SPLINE
SPL {X  -158.454, Y  +360.384, Z    +0.000, E1  +340.634, E3 -463508.318}
SPL {X  -159.737, Y  +373.507, Z    +0.000, E1  +349.689, E3 -463530.353}
SPL {X  -159.990, Y  +382.574, Z    +0.000, E1  +355.537, E3 -463537.041}
SPL {X  -159.990, Y  +389.909, Z    +0.000, E1  +360.662, E3 -463541.055}
SPL {X  -159.990, Y  +396.289, Z    +0.000, E1  +365.500, E3 -463544.835}
SPL {X  -159.990, Y  +407.941, Z    +0.000, E1  +374.126, E3 -463556.172}
SPL {X  -159.990, Y  +418.671, Z    +0.000, E1  +379.855, E3 -463575.589}
SPL {X  -159.990, Y  +429.878, Z    +0.000, E1  +383.330, E3 -463605.644}
SPL {X  -159.990, Y  +432.103, Z    +0.000, E1  +383.301, E3 -463616.662}
SPL {X  -159.990, Y  +434.188, Z    +0.000, E1  +383.325, E3 -463626.859}
SPL {X  -159.990, Y  +436.320, Z    +0.000, E1  +383.304, E3 -463637.411}
SPL {X  -159.990, Y  +439.169, Z    +0.000, E1  +383.353, E3 -463651.329}
SPL {X  -159.990, Y  +442.945, Z    +0.000, E1  +383.339, E3 -463669.946}
SPL {X  -159.990, Y  +446.037, Z    +0.000, E1  +383.324, E3 -463685.196}
SPL {X  -159.990, Y  +448.341, Z    +0.000, E1  +383.317, E3 -463696.514}
SPL {X  -159.990, Y  +450.345, Z    +0.000, E1  +383.316, E3 -463706.392}
SPL {X  -159.990, Y  +452.828, Z    +0.000, E1  +383.330, E3 -463718.591}
SPL {X  -159.990, Y  +456.338, Z    +0.000, E1  +383.359, E3 -463735.784}
SPL {X  -159.990, Y  +459.480, Z    +0.000, E1  +383.323, E3 -463751.325}
SPL {X  -159.990, Y  +461.803, Z    +0.000, E1  +383.322, E3 -463762.760}
SPL {X  -159.990, Y  +464.971, Z    +0.000, E1  +383.357, E3 -463778.266}
SPL {X  -159.990, Y  +467.934, Z    +0.000, E1  +383.321, E3 -463792.923}
SPL {X  -159.990, Y  +469.939, Z    +0.000, E1  +383.319, E3 -463802.785}
SPL {X  -159.990, Y  +472.144, Z    +0.000, E1  +383.327, E3 -463813.636}
SPL {X  -159.990, Y  +474.994, Z    +0.000, E1  +383.334, E3 -463827.684}
SPL {X  -159.990, Y  +477.323, Z    +0.000, E1  +383.307, E3 -463839.199}
SPL {X  -159.990, Y  +479.553, Z    +0.000, E1  +383.328, E3 -463850.134}
SPL {X  -159.990, Y  +482.799, Z    +0.000, E1  +383.343, E3 -463866.074}
SPL {X  -159.990, Y  +485.299, Z    +0.000, E1  +383.310, E3 -463878.459}
SPL {X  -159.990, Y  +488.031, Z    +0.000, E1  +383.345, E3 -463891.838}
SPL {X  -159.990, Y  +491.121, Z    +0.000, E1  +383.323, E3 -463907.083}
SPL {X  -159.990, Y  +493.610, Z    +0.000, E1  +383.323, E3 -463919.336}
SPL {X  -159.990, Y  +495.794, Z    +0.000, E1  +383.312, E3 -463930.110}
SPL {X  -159.990, Y  +497.668, Z    +0.000, E1  +383.317, E3 -463939.319}
SPL {X  -159.990, Y  +499.995, Z    +0.000, E1  +383.324, E3 -463950.757}
SPL {X  -159.990, Y  +502.341, Z    +0.000, E1  +383.320, E3 -463962.316}
SPL {X  -159.990, Y  +504.419, Z    +0.000, E1  +383.313, E3 -463972.558}
SPL {X  -159.990, Y  +507.187, Z    +0.000, E1  +383.346, E3 -463986.111}
SPL {X  -159.990, Y  +510.344, Z    +0.000, E1  +383.327, E3 -464001.696}
SPL {X  -159.990, Y  +512.484, Z    +0.000, E1  +383.309, E3 -464012.269}
SPL {X  -159.990, Y  +514.016, Z    +0.000, E1  +383.308, E3 -464019.817}
SPL {X  -159.990, Y  +516.195, Z    +0.000, E1  +383.325, E3 -464030.505}
SPL {X  -159.990, Y  +518.925, Z    +0.000, E1  +383.333, E3 -464043.868}
SPL {X  -159.990, Y  +521.408, Z    +0.000, E1  +383.329, E3 -464056.077}
SPL {X  -159.990, Y  +523.942, Z    +0.000, E1  +383.333, E3 -464068.570}
SPL {X  -159.990, Y  +526.221, Z    +0.000, E1  +383.314, E3 -464079.846}
SPL {X  -159.990, Y  +527.834, Z    +0.000, E1  +383.311, E3 -464087.796}
SPL {X  -159.990, Y  +529.993, Z    +0.000, E1  +383.329, E3 -464098.372}
SPL {X  -159.990, Y  +532.441, Z    +0.000, E1  +383.322, E3 -464110.423}
SPL {X  -159.990, Y  +534.618, Z    +0.000, E1  +383.322, E3 -464121.156}
SPL {X  -159.990, Y  +537.024, Z    +0.000, E1  +383.321, E3 -464133.018}
SPL {X  -159.990, Y  +539.129, Z    +0.000, E1  +383.310, E3 -464143.401}
SPL {X  -159.990, Y  +541.183, Z    +0.000, E1  +383.319, E3 -464153.498}
SPL {X  -159.990, Y  +543.647, Z    +0.000, E1  +383.325, E3 -464165.601}
SPL {X  -159.990, Y  +545.957, Z    +0.000, E1  +383.318, E3 -464176.981}
SPL {X  -159.990, Y  +548.912, Z    +0.000, E1  +383.354, E3 -464191.441}
SPL {X  -159.990, Y  +551.655, Z    +0.000, E1  +383.320, E3 -464205.016}
SPL {X  -159.990, Y  +553.711, Z    +0.000, E1  +383.317, E3 -464215.137}
SPL {X  -159.990, Y  +556.481, Z    +0.000, E1  +383.354, E3 -464228.699}
SPL {X  -159.990, Y  +559.475, Z    +0.000, E1  +383.321, E3 -464243.505}
SPL {X  -159.990, Y  +561.830, Z    +0.000, E1  +383.325, E3 -464255.089}
SPL {X  -159.990, Y  +564.273, Z    +0.000, E1  +383.325, E3 -464267.113}
SPL {X  -159.990, Y  +566.342, Z    +0.000, E1  +383.314, E3 -464277.318}
SPL {X  -159.990, Y  +568.184, Z    +0.000, E1  +383.317, E3 -464286.379}
SPL {X  -159.990, Y  +570.314, Z    +0.000, E1  +383.326, E3 -464296.841}
SPL {X  -159.990, Y  +573.444, Z    +0.000, E1  +383.356, E3 -464312.181}
SPL {X  -159.990, Y  +577.161, Z    +0.000, E1  +383.346, E3 -464330.505}
SPL {X  -159.990, Y  +580.840, Z    +0.000, E1  +383.355, E3 -464348.554}
SPL {X  -159.990, Y  +583.973, Z    +0.000, E1  +383.332, E3 -464364.016}
SPL {X  -159.990, Y  +586.020, Z    +0.000, E1  +383.323, E3 -464374.099}
SPL {X  -159.990, Y  +587.711, Z    +0.000, E1  +383.318, E3 -464382.439}
SPL {X  -159.990, Y  +589.763, Z    +0.000, E1  +383.328, E3 -464392.515}
SPL {X  -159.990, Y  +591.698, Z    +0.000, E1  +383.324, E3 -464402.000}
SPL {X  -159.990, Y  +593.847, Z    +0.000, E1  +383.340, E3 -464412.531}
SPL {X  -159.990, Y  +597.018, Z    +0.000, E1  +383.367, E3 -464428.063}
SPL {X  -159.990, Y  +599.887, Z    +0.000, E1  +383.341, E3 -464442.167}
SPL {X  -159.990, Y  +601.949, Z    +0.000, E1  +383.344, E3 -464452.294}
SPL {X  -159.990, Y  +605.106, Z    +0.000, E1  +383.383, E3 -464467.740}
SPL {X  -159.990, Y  +608.111, Z    +0.000, E1  +383.342, E3 -464482.591}
SPL {X  -159.990, Y  +610.073, Z    +0.000, E1  +383.343, E3 -464492.249}
SPL {X  -159.990, Y  +612.330, Z    +0.000, E1  +383.340, E3 -464503.376}
SPL {X  -159.990, Y  +615.036, Z    +0.000, E1  +383.353, E3 -464516.663}
SPL {X  -159.990, Y  +618.481, Z    +0.000, E1  +383.366, E3 -464533.601}
SPL {X  -159.990, Y  +621.517, Z    +0.000, E1  +383.337, E3 -464548.584}
SPL {X  -159.990, Y  +623.764, Z    +0.000, E1  +383.335, E3 -464559.635}
SPL {X  -159.990, Y  +626.608, Z    +0.000, E1  +383.361, E3 -464573.560}
SPL {X  -159.990, Y  +630.271, Z    +0.000, E1  +383.375, E3 -464591.521}
SPL {X  -159.990, Y  +633.318, Z    +0.000, E1  +383.339, E3 -464606.598}
SPL {X  -159.990, Y  +635.650, Z    +0.000, E1  +383.339, E3 -464618.069}
SPL {X  -159.990, Y  +638.406, Z    +0.000, E1  +383.354, E3 -464631.636}
SPL {X  -159.990, Y  +641.831, Z    +0.000, E1  +383.342, E3 -464648.583}
SPL {X  -159.990, Y  +644.884, Z    +0.000, E1  +383.324, E3 -464663.670}
SPL {X  -159.990, Y  +647.550, Z    +0.000, E1  +383.318, E3 -464676.837}
SPL {X  -159.990, Y  +650.790, Z    +0.000, E1  +383.346, E3 -464692.704}
SPL {X  -159.990, Y  +654.543, Z    +0.000, E1  +383.348, E3 -464711.157}
SPL {X  -159.990, Y  +658.319, Z    +0.000, E1  +383.349, E3 -464729.746}
SPL {X  -159.990, Y  +661.392, Z    +0.000, E1  +383.318, E3 -464744.949}
SPL {X  -159.990, Y  +663.662, Z    +0.000, E1  +383.322, E3 -464756.073}
SPL {X  -159.990, Y  +665.964, Z    +0.000, E1  +383.328, E3 -464767.364}
SPL {X  -159.990, Y  +667.870, Z    +0.000, E1  +383.320, E3 -464776.771}
SPL {X  -159.990, Y  +669.861, Z    +0.000, E1  +383.321, E3 -464786.572}
SPL {X  -159.983, Y  +672.946, Z    +0.000, E1  +383.359, E3 -464801.681}
SPL {X  -159.924, Y  +676.110, Z    +0.000, E1  +383.320, E3 -464817.380}
SPL {X  -159.801, Y  +679.265, Z    +0.000, E1  +383.327, E3 -464832.999}
SPL {X  -159.626, Y  +682.287, Z    +0.000, E1  +383.280, E3 -464848.097}
SPL {X  -159.462, Y  +684.486, Z    +0.000, E1  +383.258, E3 -464859.097}
SPL {X  -159.289, Y  +686.457, Z    +0.000, E1  +383.223, E3 -464869.007}
SPL {X  -159.052, Y  +688.801, Z    +0.000, E1  +383.217, E3 -464880.742}
SPL {X  -158.770, Y  +691.222, Z    +0.000, E1  +383.158, E3 -464893.000}
SPL {X  -158.553, Y  +692.896, Z    +0.000, E1  +383.130, E3 -464901.465}
ENDSPLINE

SPLINE
SPL {X  -159.063, Y  +688.696, Z    +0.000, E1  +377.094, E3 -464939.586}
SPL {X  -159.987, Y  +672.488, Z    +0.000, E1  +365.638, E3 -464963.651}
SPL {X  -159.990, Y  +663.928, Z    +0.000, E1  +359.662, E3 -464969.445}
SPL {X  -159.990, Y  +658.009, Z    +0.000, E1  +355.226, E3 -464973.145}
SPL {X  -159.990, Y  +651.879, Z    +0.000, E1  +350.548, E3 -464978.208}
SPL {X  -159.990, Y  +637.832, Z    +0.000, E1  +341.694, E3 -464995.799}
SPL {X  -159.990, Y  +626.634, Z    +0.000, E1  +337.968, E3 -465026.652}
SPL {X  -159.990, Y  +624.622, Z    +0.000, E1  +337.980, E3 -465037.235}
SPL {X  -159.990, Y  +622.489, Z    +0.000, E1  +337.969, E3 -465048.402}
SPL {X  -159.990, Y  +619.955, Z    +0.000, E1  +337.968, E3 -465061.692}
SPL {X  -159.990, Y  +617.386, Z    +0.000, E1  +337.968, E3 -465075.167}
SPL {X  -159.990, Y  +614.863, Z    +0.000, E1  +337.969, E3 -465088.399}
SPL {X  -159.990, Y  +612.600, Z    +0.000, E1  +337.975, E3 -465100.283}
SPL {X  -159.990, Y  +610.646, Z    +0.000, E1  +337.979, E3 -465110.540}
SPL {X  -159.990, Y  +608.810, Z    +0.000, E1  +337.977, E3 -465120.173}
SPL {X  -159.990, Y  +606.481, Z    +0.000, E1  +337.967, E3 -465132.349}
SPL {X  -159.990, Y  +603.419, Z    +0.000, E1  +337.936, E3 -465148.288}
SPL {X  -159.990, Y  +600.642, Z    +0.000, E1  +337.968, E3 -465162.918}
SPL {X  -159.990, Y  +598.568, Z    +0.000, E1  +337.954, E3 -465173.710}
SPL {X  -159.990, Y  +595.493, Z    +0.000, E1  +337.930, E3 -465189.794}
SPL {X  -159.990, Y  +592.865, Z    +0.000, E1  +337.964, E3 -465203.622}
SPL {X  -159.990, Y  +590.803, Z    +0.000, E1  +337.954, E3 -465214.413}
SPL {X  -159.990, Y  +588.288, Z    +0.000, E1  +337.950, E3 -465227.577}
SPL {X  -159.990, Y  +586.040, Z    +0.000, E1  +337.954, E3 -465239.322}
SPL {X  -159.990, Y  +584.080, Z    +0.000, E1  +337.953, E3 -465249.582}
SPL {X  -159.990, Y  +581.924, Z    +0.000, E1  +337.949, E3 -465260.883}
SPL {X  -159.990, Y  +579.673, Z    +0.000, E1  +337.950, E3 -465272.681}
SPL {X  -159.990, Y  +576.961, Z    +0.000, E1  +337.936, E3 -465286.860}
SPL {X  -159.990, Y  +574.188, Z    +0.000, E1  +337.947, E3 -465301.407}
SPL {X  -159.990, Y  +571.954, Z    +0.000, E1  +337.959, E3 -465313.165}
SPL {X  -159.990, Y  +570.110, Z    +0.000, E1  +337.958, E3 -465322.815}
SPL {X  -159.990, Y  +568.165, Z    +0.000, E1  +337.957, E3 -465332.995}
SPL {X  -159.990, Y  +565.292, Z    +0.000, E1  +337.922, E3 -465347.973}
SPL {X  -159.990, Y  +562.598, Z    +0.000, E1  +337.958, E3 -465362.184}
SPL {X  -159.990, Y  +560.652, Z    +0.000, E1  +337.962, E3 -465372.396}
SPL {X  -159.990, Y  +558.143, Z    +0.000, E1  +337.928, E3 -465385.428}
SPL {X  -159.990, Y  +555.329, Z    +0.000, E1  +337.943, E3 -465400.172}
SPL {X  -159.990, Y  +553.115, Z    +0.000, E1  +337.946, E3 -465411.778}
SPL {X  -159.990, Y  +550.886, Z    +0.000, E1  +337.944, E3 -465423.459}
SPL {X  -159.990, Y  +548.568, Z    +0.000, E1  +337.944, E3 -465435.580}
SPL {X  -159.990, Y  +545.859, Z    +0.000, E1  +337.926, E3 -465449.730}
SPL {X  -159.990, Y  +542.390, Z    +0.000, E1  +337.914, E3 -465467.900}
SPL {X  -159.990, Y  +539.341, Z    +0.000, E1  +337.944, E3 -465483.922}
SPL {X  -159.990, Y  +536.935, Z    +0.000, E1  +337.942, E3 -465496.511}
SPL {X  -159.990, Y  +534.656, Z    +0.000, E1  +337.946, E3 -465508.455}
SPL {X  -159.990, Y  +532.453, Z    +0.000, E1  +337.944, E3 -465519.982}
SPL {X  -159.990, Y  +530.660, Z    +0.000, E1  +337.952, E3 -465529.385}
SPL {X  -159.990, Y  +528.702, Z    +0.000, E1  +337.939, E3 -465539.598}
SPL {X  -159.990, Y  +525.760, Z    +0.000, E1  +337.914, E3 -465554.939}
SPL {X  -159.990, Y  +522.838, Z    +0.000, E1  +337.933, E3 -465570.306}
SPL {X  -159.990, Y  +519.698, Z    +0.000, E1  +337.916, E3 -465586.689}
SPL {X  -159.990, Y  +517.251, Z    +0.000, E1  +337.946, E3 -465599.549}
SPL {X  -159.990, Y  +515.568, Z    +0.000, E1  +338.084, E3 -465609.646}
ENDSPLINE

SPLINE
SPL {X  -159.990, Y  +517.293, Z    +0.000, E1  +340.923, E3 -465625.944}
ENDSPLINE

SPLINE
SPL {X  -159.990, Y  +512.548, Z    +0.000, E1  +339.587, E3 -465641.519}
SPL {X  -159.990, Y  +508.660, Z    +0.000, E1  +338.515, E3 -465653.573}
SPL {X  -159.990, Y  +503.499, Z    +0.000, E1  +337.116, E3 -465668.653}
SPL {X  -159.990, Y  +498.406, Z    +0.000, E1  +335.789, E3 -465682.685}
SPL {X  -159.990, Y  +494.693, Z    +0.000, E1  +334.929, E3 -465693.153}
SPL {X  -159.990, Y  +491.649, Z    +0.000, E1  +334.596, E3 -465704.355}
SPL {X  -159.990, Y  +488.807, Z    +0.000, E1  +334.603, E3 -465717.080}
SPL {X  -159.990, Y  +486.070, Z    +0.000, E1  +334.601, E3 -465729.311}
SPL {X  -159.990, Y  +483.747, Z    +0.000, E1  +334.616, E3 -465739.724}
SPL {X  -159.990, Y  +481.038, Z    +0.000, E1  +334.588, E3 -465751.779}
SPL {X  -159.990, Y  +478.407, Z    +0.000, E1  +334.616, E3 -465763.593}
SPL {X  -159.990, Y  +475.940, Z    +0.000, E1  +334.597, E3 -465774.583}
SPL {X  -159.990, Y  +473.026, Z    +0.000, E1  +334.601, E3 -465787.613}
SPL {X  -159.990, Y  +470.047, Z    +0.000, E1  +334.598, E3 -465800.931}
SPL {X  -159.990, Y  +467.082, Z    +0.000, E1  +334.601, E3 -465814.178}
SPL {X  -159.990, Y  +464.919, Z    +0.000, E1  +334.619, E3 -465823.905}
SPL {X  -159.990, Y  +462.520, Z    +0.000, E1  +334.600, E3 -465834.580}
SPL {X  -159.990, Y  +460.081, Z    +0.000, E1  +334.610, E3 -465845.481}
SPL {X  -159.990, Y  +457.497, Z    +0.000, E1  +334.597, E3 -465857.005}
SPL {X  -159.990, Y  +454.323, Z    +0.000, E1  +334.588, E3 -465871.165}
SPL {X  -159.990, Y  +450.823, Z    +0.000, E1  +334.583, E3 -465886.793}
SPL {X  -159.990, Y  +446.894, Z    +0.000, E1  +334.572, E3 -465904.350}
SPL {X  -159.990, Y  +443.345, Z    +0.000, E1  +334.610, E3 -465920.358}
SPL {X  -159.990, Y  +441.077, Z    +0.000, E1  +334.631, E3 -465930.556}
SPL {X  -159.990, Y  +438.608, Z    +0.000, E1  +334.608, E3 -465941.553}
SPL {X  -159.990, Y  +435.579, Z    +0.000, E1  +334.614, E3 -465955.107}
SPL {X  -159.990, Y  +432.613, Z    +0.000, E1  +334.610, E3 -465968.374}
SPL {X  -159.990, Y  +429.079, Z    +0.000, E1  +334.593, E3 -465984.145}
SPL {X  -159.990, Y  +426.149, Z    +0.000, E1  +334.626, E3 -465997.307}
SPL {X  -159.990, Y  +423.417, Z    +0.000, E1  +334.600, E3 -466009.472}
SPL {X  -159.990, Y  +419.467, Z    +0.000, E1  +334.583, E3 -466027.107}
SPL {X  -159.990, Y  +415.368, Z    +0.000, E1  +334.593, E3 -466045.462}
SPL {X  -159.990, Y  +411.297, Z    +0.000, E1  +334.587, E3 -466063.657}
SPL {X  -159.990, Y  +407.450, Z    +0.000, E1  +334.599, E3 -466080.871}
SPL {X  -159.990, Y  +403.513, Z    +0.000, E1  +334.580, E3 -466098.425}
SPL {X  -159.990, Y  +399.294, Z    +0.000, E1  +334.582, E3 -466117.305}
SPL {X  -159.990, Y  +395.411, Z    +0.000, E1  +334.600, E3 -466134.719}
SPL {X  -159.990, Y  +392.473, Z    +0.000, E1  +334.623, E3 -466147.904}
SPL {X  -159.990, Y  +390.187, Z    +0.000, E1  +334.622, E3 -466158.163}
SPL {X  -159.990, Y  +387.503, Z    +0.000, E1  +334.622, E3 -466170.157}
SPL {X  -159.990, Y  +384.711, Z    +0.000, E1  +334.612, E3 -466182.601}
SPL {X  -159.988, Y  +381.794, Z    +0.000, E1  +334.611, E3 -466195.636}
SPL {X  -159.958, Y  +379.279, Z    +0.000, E1  +334.625, E3 -466206.926}
SPL {X  -159.894, Y  +376.959, Z    +0.000, E1  +334.630, E3 -466217.370}
SPL {X  -159.765, Y  +374.027, Z    +0.000, E1  +334.633, E3 -466230.586}
SPL {X  -159.607, Y  +371.442, Z    +0.000, E1  +334.673, E3 -466242.361}
SPL {X  -159.379, Y  +368.534, Z    +0.000, E1  +334.684, E3 -466255.549}
SPL {X  -159.113, Y  +365.767, Z    +0.000, E1  +334.734, E3 -466268.188}
SPL {X  -158.869, Y  +363.595, Z    +0.000, E1  +334.770, E3 -466278.160}
SPL {X  -158.527, Y  +360.915, Z    +0.000, E1  +334.798, E3 -466290.466}
SPL {X  -158.127, Y  +358.155, Z    +0.000, E1  +334.874, E3 -466303.304}
SPL {X  -158.095, Y  +357.947, Z    +0.000, E1  +338.259, E3 -466334.876}
ENDSPLINE

SPLINE
SPL {X  -158.454, Y  +360.384, Z    +0.000, E1  +340.634, E3 -466347.027}
SPL {X  -159.737, Y  +373.507, Z    +0.000, E1  +349.689, E3 -466369.063}
SPL {X  -159.990, Y  +382.574, Z    +0.000, E1  +355.537, E3 -466375.750}
SPL {X  -159.990, Y  +387.496, Z    +0.000, E1  +358.996, E3 -466378.496}
SPL {X  -159.990, Y  +395.121, Z    +0.000, E1  +364.514, E3 -466382.808}
SPL {X  -159.990, Y  +407.941, Z    +0.000, E1  +374.126, E3 -466394.882}
SPL {X  -159.990, Y  +418.671, Z    +0.000, E1  +379.855, E3 -466414.298}
SPL {X  -159.990, Y  +429.878, Z    +0.000, E1  +383.330, E3 -466444.353}
SPL {X  -159.990, Y  +432.103, Z    +0.000, E1  +383.301, E3 -466455.372}
SPL {X  -159.990, Y  +434.188, Z    +0.000, E1  +383.325, E3 -466465.568}
SPL {X  -159.990, Y  +436.320, Z    +0.000, E1  +383.304, E3 -466476.121}
SPL {X  -159.990, Y  +439.169, Z    +0.000, E1  +383.353, E3 -466490.038}
SPL {X  -159.990, Y  +442.945, Z    +0.000, E1  +383.339, E3 -466508.656}
SPL {X  -159.990, Y  +446.037, Z    +0.000, E1  +383.324, E3 -466523.906}
SPL {X  -159.990, Y  +448.341, Z    +0.000, E1  +383.317, E3 -466535.224}
SPL {X  -159.990, Y  +450.968, Z    +0.000, E1  +383.336, E3 -466548.139}
SPL {X  -159.990, Y  +454.421, Z    +0.000, E1  +383.348, E3 -466565.088}
SPL {X  -159.990, Y  +457.167, Z    +0.000, E1  +383.324, E3 -466578.631}
SPL {X  -159.990, Y  +459.480, Z    +0.000, E1  +383.323, E3 -466590.035}
SPL {X  -159.990, Y  +462.520, Z    +0.000, E1  +383.350, E3 -466604.939}
SPL {X  -159.990, Y  +465.602, Z    +0.000, E1  +383.328, E3 -466620.139}
SPL {X  -159.990, Y  +467.934, Z    +0.000, E1  +383.321, E3 -466631.633}
SPL {X  -159.990, Y  +469.939, Z    +0.000, E1  +383.319, E3 -466641.495}
SPL {X  -159.990, Y  +472.144, Z    +0.000, E1  +383.327, E3 -466652.345}
SPL {X  -159.990, Y  +474.152, Z    +0.000, E1  +383.309, E3 -466662.297}
SPL {X  -159.990, Y  +476.560, Z    +0.000, E1  +383.332, E3 -466674.106}
SPL {X  -159.990, Y  +478.770, Z    +0.000, E1  +383.306, E3 -466685.031}
SPL {X  -159.990, Y  +480.905, Z    +0.000, E1  +383.327, E3 -466695.499}
SPL {X  -159.990, Y  +484.251, Z    +0.000, E1  +383.352, E3 -466711.914}
SPL {X  -159.990, Y  +488.031, Z    +0.000, E1  +383.345, E3 -466730.547}
SPL {X  -159.990, Y  +491.121, Z    +0.000, E1  +383.323, E3 -466745.793}
SPL {X  -159.990, Y  +493.610, Z    +0.000, E1  +383.323, E3 -466758.046}
SPL {X  -159.990, Y  +496.863, Z    +0.000, E1  +383.350, E3 -466774.006}
SPL {X  -159.990, Y  +499.995, Z    +0.000, E1  +383.324, E3 -466789.467}
SPL {X  -159.990, Y  +502.341, Z    +0.000, E1  +383.320, E3 -466801.026}
SPL {X  -159.990, Y  +505.377, Z    +0.000, E1  +383.346, E3 -466815.917}
SPL {X  -159.990, Y  +508.024, Z    +0.000, E1  +383.315, E3 -466828.999}
SPL {X  -159.990, Y  +510.344, Z    +0.000, E1  +383.327, E3 -466840.406}
SPL {X  -159.990, Y  +513.289, Z    +0.000, E1  +383.332, E3 -466854.896}
SPL {X  -159.990, Y  +516.195, Z    +0.000, E1  +383.325, E3 -466869.215}
SPL {X  -159.990, Y  +518.925, Z    +0.000, E1  +383.333, E3 -466882.578}
SPL {X  -159.990, Y  +521.408, Z    +0.000, E1  +383.329, E3 -466894.787}
SPL {X  -159.990, Y  +523.942, Z    +0.000, E1  +383.333, E3 -466907.280}
SPL {X  -159.990, Y  +526.221, Z    +0.000, E1  +383.314, E3 -466918.556}
SPL {X  -159.990, Y  +527.834, Z    +0.000, E1  +383.311, E3 -466926.506}
SPL {X  -159.990, Y  +529.993, Z    +0.000, E1  +383.329, E3 -466937.082}
SPL {X  -159.990, Y  +532.441, Z    +0.000, E1  +383.322, E3 -466949.133}
SPL {X  -159.990, Y  +534.618, Z    +0.000, E1  +383.322, E3 -466959.866}
SPL {X  -159.990, Y  +537.024, Z    +0.000, E1  +383.321, E3 -466971.728}
SPL {X  -159.990, Y  +539.129, Z    +0.000, E1  +383.310, E3 -466982.111}
SPL {X  -159.990, Y  +541.183, Z    +0.000, E1  +383.319, E3 -466992.208}
SPL {X  -159.990, Y  +543.647, Z    +0.000, E1  +383.325, E3 -467004.311}
SPL {X  -159.990, Y  +546.832, Z    +0.000, E1  +383.349, E3 -467019.933}
SPL {X  -159.990, Y  +549.756, Z    +0.000, E1  +383.320, E3 -467034.374}
SPL {X  -159.990, Y  +551.655, Z    +0.000, E1  +383.320, E3 -467043.725}
SPL {X  -159.990, Y  +553.711, Z    +0.000, E1  +383.317, E3 -467053.847}
SPL {X  -159.990, Y  +555.637, Z    +0.000, E1  +383.323, E3 -467063.316}
SPL {X  -159.990, Y  +558.758, Z    +0.000, E1  +383.351, E3 -467078.626}
SPL {X  -159.990, Y  +561.830, Z    +0.000, E1  +383.325, E3 -467093.799}
SPL {X  -159.990, Y  +564.273, Z    +0.000, E1  +383.325, E3 -467105.823}
SPL {X  -159.990, Y  +567.351, Z    +0.000, E1  +383.348, E3 -467120.919}
SPL {X  -159.990, Y  +570.314, Z    +0.000, E1  +383.326, E3 -467135.551}
SPL {X  -159.990, Y  +572.504, Z    +0.000, E1  +383.321, E3 -467146.336}
SPL {X  -159.990, Y  +575.653, Z    +0.000, E1  +383.355, E3 -467161.773}
SPL {X  -159.990, Y  +578.932, Z    +0.000, E1  +383.330, E3 -467177.955}
SPL {X  -159.990, Y  +581.497, Z    +0.000, E1  +383.329, E3 -467190.540}
SPL {X  -159.990, Y  +583.973, Z    +0.000, E1  +383.332, E3 -467202.725}
SPL {X  -159.990, Y  +586.020, Z    +0.000, E1  +383.323, E3 -467212.809}
SPL {X  -159.990, Y  +587.711, Z    +0.000, E1  +383.318, E3 -467221.149}
SPL {X  -159.990, Y  +589.763, Z    +0.000, E1  +383.328, E3 -467231.225}
SPL {X  -159.990, Y  +591.698, Z    +0.000, E1  +383.324, E3 -467240.710}
SPL {X  -159.990, Y  +593.847, Z    +0.000, E1  +383.340, E3 -467251.240}
SPL {X  -159.990, Y  +597.018, Z    +0.000, E1  +383.367, E3 -467266.772}
SPL {X  -159.990, Y  +599.887, Z    +0.000, E1  +383.341, E3 -467280.877}
SPL {X  -159.990, Y  +601.949, Z    +0.000, E1  +383.344, E3 -467291.003}
SPL {X  -159.990, Y  +605.106, Z    +0.000, E1  +383.383, E3 -467306.449}
SPL {X  -159.990, Y  +608.111, Z    +0.000, E1  +383.342, E3 -467321.300}
SPL {X  -159.990, Y  +610.073, Z    +0.000, E1  +383.343, E3 -467330.958}
SPL {X  -159.990, Y  +612.330, Z    +0.000, E1  +383.340, E3 -467342.086}
SPL {X  -159.990, Y  +615.036, Z    +0.000, E1  +383.353, E3 -467355.373}
SPL {X  -159.990, Y  +618.481, Z    +0.000, E1  +383.366, E3 -467372.311}
SPL {X  -159.990, Y  +621.517, Z    +0.000, E1  +383.337, E3 -467387.294}
SPL {X  -159.990, Y  +623.764, Z    +0.000, E1  +383.335, E3 -467398.345}
SPL {X  -159.990, Y  +626.608, Z    +0.000, E1  +383.361, E3 -467412.269}
SPL {X  -159.990, Y  +630.271, Z    +0.000, E1  +383.375, E3 -467430.231}
SPL {X  -159.990, Y  +633.318, Z    +0.000, E1  +383.339, E3 -467445.308}
SPL {X  -159.990, Y  +635.650, Z    +0.000, E1  +383.339, E3 -467456.779}
SPL {X  -159.990, Y  +638.406, Z    +0.000, E1  +383.354, E3 -467470.346}
SPL {X  -159.990, Y  +641.831, Z    +0.000, E1  +383.342, E3 -467487.293}
SPL {X  -159.990, Y  +644.884, Z    +0.000, E1  +383.324, E3 -467502.380}
SPL {X  -159.990, Y  +647.550, Z    +0.000, E1  +383.318, E3 -467515.547}
SPL {X  -159.990, Y  +650.790, Z    +0.000, E1  +383.346, E3 -467531.413}
SPL {X  -159.990, Y  +654.543, Z    +0.000, E1  +383.348, E3 -467549.866}
SPL {X  -159.990, Y  +658.319, Z    +0.000, E1  +383.349, E3 -467568.456}
SPL {X  -159.990, Y  +661.392, Z    +0.000, E1  +383.318, E3 -467583.659}
SPL {X  -159.990, Y  +663.662, Z    +0.000, E1  +383.322, E3 -467594.783}
SPL {X  -159.990, Y  +665.964, Z    +0.000, E1  +383.328, E3 -467606.074}
SPL {X  -159.990, Y  +667.870, Z    +0.000, E1  +383.320, E3 -467615.480}
SPL {X  -159.990, Y  +669.861, Z    +0.000, E1  +383.321, E3 -467625.282}
SPL {X  -159.990, Y  +671.893, Z    +0.000, E1  +383.319, E3 -467635.289}
SPL {X  -159.974, Y  +673.789, Z    +0.000, E1  +383.323, E3 -467644.605}
SPL {X  -159.924, Y  +676.110, Z    +0.000, E1  +383.320, E3 -467656.090}
SPL {X  -159.801, Y  +679.265, Z    +0.000, E1  +383.327, E3 -467671.708}
SPL {X  -159.626, Y  +682.287, Z    +0.000, E1  +383.280, E3 -467686.807}
SPL {X  -159.462, Y  +684.486, Z    +0.000, E1  +383.258, E3 -467697.807}
SPL {X  -159.212, Y  +687.262, Z    +0.000, E1  +383.238, E3 -467711.710}
SPL {X  -158.971, Y  +689.529, Z    +0.000, E1  +383.181, E3 -467723.170}
SPL {X  -158.658, Y  +692.098, Z    +0.000, E1  +383.176, E3 -467736.077}
ENDSPLINE

SPLINE
SPL {X  -159.063, Y  +688.696, Z    +0.000, E1  +377.094, E3 -467778.295}
SPL {X  -159.957, Y  +674.769, Z    +0.000, E1  +367.092, E3 -467800.677}
SPL {X  -159.990, Y  +671.516, Z    +0.000, E1  +364.944, E3 -467803.063}
SPL {X  -159.990, Y  +663.928, Z    +0.000, E1  +359.662, E3 -467808.155}
SPL {X  -159.990, Y  +658.009, Z    +0.000, E1  +355.226, E3 -467811.855}
SPL {X  -159.990, Y  +651.879, Z    +0.000, E1  +350.548, E3 -467816.917}
SPL {X  -159.990, Y  +637.832, Z    +0.000, E1  +341.694, E3 -467834.508}
SPL {X  -159.990, Y  +626.634, Z    +0.000, E1  +337.968, E3 -467865.361}
SPL {X  -159.990, Y  +624.622, Z    +0.000, E1  +337.980, E3 -467875.945}
SPL {X  -159.990, Y  +622.489, Z    +0.000, E1  +337.969, E3 -467887.111}
SPL {X  -159.990, Y  +619.955, Z    +0.000, E1  +337.968, E3 -467900.401}
SPL {X  -159.990, Y  +617.386, Z    +0.000, E1  +337.968, E3 -467913.876}
SPL {X  -159.990, Y  +614.863, Z    +0.000, E1  +337.969, E3 -467927.108}
SPL {X  -159.990, Y  +612.600, Z    +0.000, E1  +337.975, E3 -467938.993}
SPL {X  -159.990, Y  +610.646, Z    +0.000, E1  +337.979, E3 -467949.250}
SPL {X  -159.990, Y  +608.810, Z    +0.000, E1  +337.977, E3 -467958.883}
SPL {X  -159.990, Y  +605.804, Z    +0.000, E1  +337.936, E3 -467974.528}
SPL {X  -159.990, Y  +602.819, Z    +0.000, E1  +337.963, E3 -467990.199}
SPL {X  -159.990, Y  +600.642, Z    +0.000, E1  +337.968, E3 -468001.627}
SPL {X  -159.990, Y  +598.568, Z    +0.000, E1  +337.954, E3 -468012.420}
SPL {X  -159.990, Y  +596.440, Z    +0.000, E1  +337.964, E3 -468023.602}
SPL {X  -159.990, Y  +593.768, Z    +0.000, E1  +337.929, E3 -468037.535}
SPL {X  -159.990, Y  +590.803, Z    +0.000, E1  +337.954, E3 -468053.123}
SPL {X  -159.990, Y  +588.288, Z    +0.000, E1  +337.950, E3 -468066.287}
SPL {X  -159.990, Y  +586.040, Z    +0.000, E1  +337.954, E3 -468078.032}
SPL {X  -159.990, Y  +584.080, Z    +0.000, E1  +337.953, E3 -468088.292}
SPL {X  -159.990, Y  +581.924, Z    +0.000, E1  +337.949, E3 -468099.592}
SPL {X  -159.990, Y  +579.673, Z    +0.000, E1  +337.950, E3 -468111.390}
SPL {X  -159.990, Y  +576.961, Z    +0.000, E1  +337.936, E3 -468125.570}
SPL {X  -159.990, Y  +574.188, Z    +0.000, E1  +337.947, E3 -468140.117}
SPL {X  -159.990, Y  +571.954, Z    +0.000, E1  +337.959, E3 -468151.875}
SPL {X  -159.990, Y  +570.110, Z    +0.000, E1  +337.958, E3 -468161.525}
SPL {X  -159.990, Y  +568.165, Z    +0.000, E1  +337.957, E3 -468171.705}
SPL {X  -159.990, Y  +565.292, Z    +0.000, E1  +337.922, E3 -468186.683}
SPL {X  -159.990, Y  +562.598, Z    +0.000, E1  +337.958, E3 -468200.894}
SPL {X  -159.990, Y  +560.652, Z    +0.000, E1  +337.962, E3 -468211.106}
SPL {X  -159.990, Y  +558.143, Z    +0.000, E1  +337.928, E3 -468224.138}
SPL {X  -159.990, Y  +555.329, Z    +0.000, E1  +337.943, E3 -468238.882}
SPL {X  -159.990, Y  +553.115, Z    +0.000, E1  +337.946, E3 -468250.487}
SPL {X  -159.990, Y  +550.886, Z    +0.000, E1  +337.944, E3 -468262.169}
SPL {X  -159.990, Y  +548.568, Z    +0.000, E1  +337.944, E3 -468274.290}
SPL {X  -159.990, Y  +546.537, Z    +0.000, E1  +337.948, E3 -468284.925}
SPL {X  -159.990, Y  +545.062, Z    +0.000, E1  +337.955, E3 -468292.683}
SPL {X  -159.990, Y  +543.060, Z    +0.000, E1  +337.943, E3 -468303.163}
SPL {X  -159.990, Y  +539.928, Z    +0.000, E1  +337.917, E3 -468319.504}
SPL {X  -159.990, Y  +536.935, Z    +0.000, E1  +337.942, E3 -468335.221}
SPL {X  -159.990, Y  +534.656, Z    +0.000, E1  +337.946, E3 -468347.165}
SPL {X  -159.990, Y  +531.679, Z    +0.000, E1  +337.913, E3 -468362.679}
SPL {X  -159.990, Y  +527.941, Z    +0.000, E1  +337.907, E3 -468382.221}
SPL {X  -159.990, Y  +525.053, Z    +0.000, E1  +337.942, E3 -468397.411}
SPL {X  -159.990, Y  +522.838, Z    +0.000, E1  +337.933, E3 -468409.015}
SPL {X  -159.990, Y  +519.698, Z    +0.000, E1  +337.916, E3 -468425.398}
SPL {X  -159.990, Y  +517.251, Z    +0.000, E1  +337.946, E3 -468438.258}
SPL {X  -159.990, Y  +515.568, Z    +0.000, E1  +338.084, E3 -468448.355}
ENDSPLINE

SPLINE
SPL {X  -159.990, Y  +518.374, Z    +0.000, E1  +341.240, E3 -468460.943}
ENDSPLINE

SPLINE
SPL {X  -159.990, Y  +513.606, Z    +0.000, E1  +339.879, E3 -468476.854}
SPL {X  -159.990, Y  +508.660, Z    +0.000, E1  +338.515, E3 -468492.283}
SPL {X  -159.990, Y  +505.237, Z    +0.000, E1  +337.606, E3 -468502.540}
SPL {X  -159.990, Y  +501.963, Z    +0.000, E1  +336.712, E3 -468511.644}
SPL {X  -159.990, Y  +498.406, Z    +0.000, E1  +335.789, E3 -468521.395}
SPL {X  -159.990, Y  +494.693, Z    +0.000, E1  +334.929, E3 -468531.863}
SPL {X  -159.990, Y  +491.649, Z    +0.000, E1  +334.596, E3 -468543.065}
SPL {X  -159.990, Y  +488.807, Z    +0.000, E1  +334.603, E3 -468555.789}
SPL {X  -159.990, Y  +486.070, Z    +0.000, E1  +334.601, E3 -468568.020}
SPL {X  -159.990, Y  +482.821, Z    +0.000, E1  +334.589, E3 -468582.522}
SPL {X  -159.990, Y  +479.252, Z    +0.000, E1  +334.588, E3 -468598.473}
SPL {X  -159.990, Y  +475.940, Z    +0.000, E1  +334.597, E3 -468613.293}
SPL {X  -159.990, Y  +473.026, Z    +0.000, E1  +334.601, E3 -468626.323}
SPL {X  -159.990, Y  +470.047, Z    +0.000, E1  +334.598, E3 -468639.641}
SPL {X  -159.990, Y  +466.213, Z    +0.000, E1  +334.567, E3 -468656.721}
SPL {X  -159.990, Y  +462.520, Z    +0.000, E1  +334.600, E3 -468673.289}
SPL {X  -159.990, Y  +460.081, Z    +0.000, E1  +334.610, E3 -468684.191}
SPL {X  -159.990, Y  +457.497, Z    +0.000, E1  +334.597, E3 -468695.715}
SPL {X  -159.990, Y  +455.126, Z    +0.000, E1  +334.611, E3 -468706.324}
SPL {X  -159.990, Y  +453.438, Z    +0.000, E1  +334.615, E3 -468713.883}
SPL {X  -159.990, Y  +450.823, Z    +0.000, E1  +334.583, E3 -468725.503}
SPL {X  -159.990, Y  +447.982, Z    +0.000, E1  +334.607, E3 -468738.244}
SPL {X  -159.990, Y  +445.108, Z    +0.000, E1  +334.593, E3 -468751.121}
SPL {X  -159.990, Y  +441.797, Z    +0.000, E1  +334.610, E3 -468766.000}
SPL {X  -159.990, Y  +438.608, Z    +0.000, E1  +334.608, E3 -468780.262}
SPL {X  -159.990, Y  +434.852, Z    +0.000, E1  +334.585, E3 -468797.017}
SPL {X  -159.990, Y  +431.966, Z    +0.000, E1  +334.629, E3 -468810.015}
SPL {X  -159.990, Y  +429.079, Z    +0.000, E1  +334.593, E3 -468822.855}
SPL {X  -159.990, Y  +426.149, Z    +0.000, E1  +334.626, E3 -468836.017}
SPL {X  -159.990, Y  +423.417, Z    +0.000, E1  +334.600, E3 -468848.182}
SPL {X  -159.990, Y  +420.283, Z    +0.000, E1  +334.614, E3 -468862.226}
SPL {X  -159.990, Y  +417.103, Z    +0.000, E1  +334.600, E3 -468876.422}
SPL {X  -159.990, Y  +413.684, Z    +0.000, E1  +334.603, E3 -468891.721}
SPL {X  -159.990, Y  +410.645, Z    +0.000, E1  +334.615, E3 -468905.333}
SPL {X  -159.990, Y  +407.450, Z    +0.000, E1  +334.599, E3 -468919.581}
SPL {X  -159.990, Y  +404.255, Z    +0.000, E1  +334.609, E3 -468933.872}
SPL {X  -159.990, Y  +401.103, Z    +0.000, E1  +334.596, E3 -468947.936}
SPL {X  -159.990, Y  +397.743, Z    +0.000, E1  +334.600, E3 -468962.986}
SPL {X  -159.990, Y  +394.848, Z    +0.000, E1  +334.621, E3 -468975.987}
SPL {X  -159.990, Y  +392.473, Z    +0.000, E1  +334.623, E3 -468986.614}
SPL {X  -159.990, Y  +390.187, Z    +0.000, E1  +334.622, E3 -468996.872}
SPL {X  -159.990, Y  +387.503, Z    +0.000, E1  +334.622, E3 -469008.867}
SPL {X  -159.990, Y  +384.711, Z    +0.000, E1  +334.612, E3 -469021.311}
SPL {X  -159.988, Y  +381.794, Z    +0.000, E1  +334.611, E3 -469034.346}
SPL {X  -159.958, Y  +379.279, Z    +0.000, E1  +334.625, E3 -469045.636}
SPL {X  -159.894, Y  +376.959, Z    +0.000, E1  +334.630, E3 -469056.080}
SPL {X  -159.765, Y  +374.027, Z    +0.000, E1  +334.633, E3 -469069.296}
SPL {X  -159.607, Y  +371.442, Z    +0.000, E1  +334.673, E3 -469081.071}
SPL {X  -159.379, Y  +368.534, Z    +0.000, E1  +334.684, E3 -469094.258}
SPL {X  -159.113, Y  +365.767, Z    +0.000, E1  +334.734, E3 -469106.898}
SPL {X  -158.798, Y  +363.007, Z    +0.000, E1  +334.761, E3 -469119.538}
SPL {X  -158.453, Y  +360.380, Z    +0.000, E1  +334.828, E3 -469131.683}
SPL {X  -158.127, Y  +358.155, Z    +0.000, E1  +334.874, E3 -469142.013}
SPL {X  -158.095, Y  +357.947, Z    +0.000, E1  +338.259, E3 -469173.586}
ENDSPLINE

SPLINE
SPL {X  -158.454, Y  +360.384, Z    +0.000, E1  +340.634, E3 -469185.737}
SPL {X  -159.737, Y  +373.507, Z    +0.000, E1  +349.689, E3 -469207.772}
SPL {X  -159.990, Y  +382.574, Z    +0.000, E1  +355.537, E3 -469214.460}
SPL {X  -159.990, Y  +389.909, Z    +0.000, E1  +360.662, E3 -469218.475}
SPL {X  -159.990, Y  +396.289, Z    +0.000, E1  +365.500, E3 -469222.255}
SPL {X  -159.990, Y  +407.941, Z    +0.000, E1  +374.126, E3 -469233.592}
SPL {X  -159.990, Y  +418.671, Z    +0.000, E1  +379.855, E3 -469253.008}
SPL {X  -159.990, Y  +429.878, Z    +0.000, E1  +383.330, E3 -469283.063}
SPL {X  -159.990, Y  +432.766, Z    +0.000, E1  +383.321, E3 -469297.286}
SPL {X  -159.990, Y  +434.794, Z    +0.000, E1  +383.304, E3 -469307.317}
SPL {X  -159.990, Y  +437.007, Z    +0.000, E1  +383.323, E3 -469318.169}
SPL {X  -159.990, Y  +439.778, Z    +0.000, E1  +383.323, E3 -469331.802}
SPL {X  -159.990, Y  +442.010, Z    +0.000, E1  +383.308, E3 -469342.823}
SPL {X  -159.990, Y  +443.729, Z    +0.000, E1  +383.310, E3 -469351.279}
SPL {X  -159.990, Y  +446.037, Z    +0.000, E1  +383.324, E3 -469362.616}
SPL {X  -159.990, Y  +448.341, Z    +0.000, E1  +383.317, E3 -469373.933}
SPL {X  -159.990, Y  +450.345, Z    +0.000, E1  +383.316, E3 -469383.811}
SPL {X  -159.990, Y  +452.828, Z    +0.000, E1  +383.330, E3 -469396.011}
SPL {X  -159.990, Y  +456.338, Z    +0.000, E1  +383.359, E3 -469413.203}
SPL {X  -159.990, Y  +459.480, Z    +0.000, E1  +383.323, E3 -469428.744}
SPL {X  -159.990, Y  +461.803, Z    +0.000, E1  +383.322, E3 -469440.179}
SPL {X  -159.990, Y  +464.971, Z    +0.000, E1  +383.357, E3 -469455.685}
SPL {X  -159.990, Y  +467.934, Z    +0.000, E1  +383.321, E3 -469470.343}
SPL {X  -159.990, Y  +469.939, Z    +0.000, E1  +383.319, E3 -469480.204}
SPL {X  -159.990, Y  +472.144, Z    +0.000, E1  +383.327, E3 -469491.055}
SPL {X  -159.990, Y  +474.152, Z    +0.000, E1  +383.309, E3 -469501.007}
SPL {X  -159.990, Y  +476.560, Z    +0.000, E1  +383.332, E3 -469512.815}
SPL {X  -159.990, Y  +478.770, Z    +0.000, E1  +383.306, E3 -469523.740}
SPL {X  -159.990, Y  +480.905, Z    +0.000, E1  +383.327, E3 -469534.208}
SPL {X  -159.990, Y  +484.251, Z    +0.000, E1  +383.352, E3 -469550.624}
SPL {X  -159.990, Y  +488.031, Z    +0.000, E1  +383.345, E3 -469569.257}
SPL {X  -159.990, Y  +491.121, Z    +0.000, E1  +383.323, E3 -469584.502}
SPL {X  -159.990, Y  +493.610, Z    +0.000, E1  +383.323, E3 -469596.755}
SPL {X  -159.990, Y  +496.863, Z    +0.000, E1  +383.350, E3 -469612.715}
SPL {X  -159.990, Y  +499.995, Z    +0.000, E1  +383.324, E3 -469628.177}
SPL {X  -159.990, Y  +502.341, Z    +0.000, E1  +383.320, E3 -469639.736}
SPL {X  -159.990, Y  +504.419, Z    +0.000, E1  +383.313, E3 -469649.977}
SPL {X  -159.990, Y  +507.187, Z    +0.000, E1  +383.346, E3 -469663.530}
SPL {X  -159.990, Y  +510.344, Z    +0.000, E1  +383.327, E3 -469679.115}
SPL {X  -159.990, Y  +512.484, Z    +0.000, E1  +383.309, E3 -469689.688}
SPL {X  -159.990, Y  +514.016, Z    +0.000, E1  +383.308, E3 -469697.237}
SPL {X  -159.990, Y  +516.195, Z    +0.000, E1  +383.325, E3 -469707.924}
SPL {X  -159.990, Y  +518.925, Z    +0.000, E1  +383.333, E3 -469721.288}
SPL {X  -159.990, Y  +521.408, Z    +0.000, E1  +383.329, E3 -469733.497}
SPL {X  -159.990, Y  +523.942, Z    +0.000, E1  +383.333, E3 -469745.990}
SPL {X  -159.990, Y  +527.007, Z    +0.000, E1  +383.339, E3 -469761.089}
SPL {X  -159.990, Y  +529.993, Z    +0.000, E1  +383.329, E3 -469775.791}
SPL {X  -159.990, Y  +532.441, Z    +0.000, E1  +383.322, E3 -469787.842}
SPL {X  -159.990, Y  +534.618, Z    +0.000, E1  +383.322, E3 -469798.575}
SPL {X  -159.990, Y  +537.024, Z    +0.000, E1  +383.321, E3 -469810.438}
SPL {X  -159.990, Y  +539.129, Z    +0.000, E1  +383.310, E3 -469820.821}
SPL {X  -159.990, Y  +541.183, Z    +0.000, E1  +383.319, E3 -469830.917}
SPL {X  -159.990, Y  +543.647, Z    +0.000, E1  +383.325, E3 -469843.020}
SPL {X  -159.990, Y  +545.957, Z    +0.000, E1  +383.318, E3 -469854.400}
SPL {X  -159.990, Y  +548.912, Z    +0.000, E1  +383.354, E3 -469868.860}
SPL {X  -159.990, Y  +551.655, Z    +0.000, E1  +383.320, E3 -469882.435}
SPL {X  -159.990, Y  +553.711, Z    +0.000, E1  +383.317, E3 -469892.557}
SPL {X  -159.990, Y  +556.481, Z    +0.000, E1  +383.354, E3 -469906.118}
SPL {X  -159.990, Y  +559.475, Z    +0.000, E1  +383.321, E3 -469920.924}
SPL {X  -159.990, Y  +561.830, Z    +0.000, E1  +383.325, E3 -469932.508}
SPL {X  -159.990, Y  +564.273, Z    +0.000, E1  +383.325, E3 -469944.533}
SPL {X  -159.990, Y  +566.342, Z    +0.000, E1  +383.314, E3 -469954.737}
SPL {X  -159.990, Y  +568.184, Z    +0.000, E1  +383.317, E3 -469963.798}
SPL {X  -159.990, Y  +570.314, Z    +0.000, E1  +383.326, E3 -469974.261}
SPL {X  -159.990, Y  +573.444, Z    +0.000, E1  +383.356, E3 -469989.600}
SPL {X  -159.990, Y  +577.161, Z    +0.000, E1  +383.346, E3 -470007.924}
SPL {X  -159.990, Y  +580.840, Z    +0.000, E1  +383.355, E3 -470025.974}
SPL {X  -159.990, Y  +583.973, Z    +0.000, E1  +383.332, E3 -470041.435}
SPL {X  -159.990, Y  +586.020, Z    +0.000, E1  +383.323, E3 -470051.519}
SPL {X  -159.990, Y  +587.711, Z    +0.000, E1  +383.318, E3 -470059.858}
SPL {X  -159.990, Y  +589.763, Z    +0.000, E1  +383.328, E3 -470069.935}
SPL {X  -159.990, Y  +591.698, Z    +0.000, E1  +383.324, E3 -470079.419}
SPL {X  -159.990, Y  +593.847, Z    +0.000, E1  +383.340, E3 -470089.950}
SPL {X  -159.990, Y  +597.018, Z    +0.000, E1  +383.367, E3 -470105.482}
SPL {X  -159.990, Y  +599.887, Z    +0.000, E1  +383.341, E3 -470119.586}
SPL {X  -159.990, Y  +601.949, Z    +0.000, E1  +383.344, E3 -470129.713}
SPL {X  -159.990, Y  +605.106, Z    +0.000, E1  +383.383, E3 -470145.159}
SPL {X  -159.990, Y  +608.111, Z    +0.000, E1  +383.342, E3 -470160.010}
SPL {X  -159.990, Y  +610.073, Z    +0.000, E1  +383.343, E3 -470169.668}
SPL {X  -159.990, Y  +613.021, Z    +0.000, E1  +383.365, E3 -470184.139}
SPL {X  -159.990, Y  +615.657, Z    +0.000, E1  +383.331, E3 -470197.187}
SPL {X  -159.990, Y  +617.658, Z    +0.000, E1  +383.335, E3 -470207.029}
SPL {X  -159.990, Y  +620.788, Z    +0.000, E1  +383.368, E3 -470222.362}
SPL {X  -159.990, Y  +624.347, Z    +0.000, E1  +383.355, E3 -470239.882}
SPL {X  -159.990, Y  +627.144, Z    +0.000, E1  +383.340, E3 -470253.652}
SPL {X  -159.990, Y  +629.284, Z    +0.000, E1  +383.339, E3 -470264.160}
SPL {X  -159.990, Y  +631.206, Z    +0.000, E1  +383.337, E3 -470273.613}
SPL {X  -159.990, Y  +633.318, Z    +0.000, E1  +383.339, E3 -470284.018}
SPL {X  -159.990, Y  +635.650, Z    +0.000, E1  +383.339, E3 -470295.489}
SPL {X  -159.990, Y  +637.597, Z    +0.000, E1  +383.330, E3 -470305.111}
SPL {X  -159.990, Y  +640.369, Z    +0.000, E1  +383.354, E3 -470318.746}
SPL {X  -159.990, Y  +644.241, Z    +0.000, E1  +383.355, E3 -470337.858}
SPL {X  -159.990, Y  +648.287, Z    +0.000, E1  +383.349, E3 -470357.814}
SPL {X  -159.990, Y  +651.427, Z    +0.000, E1  +383.319, E3 -470373.310}
SPL {X  -159.990, Y  +653.536, Z    +0.000, E1  +383.313, E3 -470383.691}
SPL {X  -159.990, Y  +656.380, Z    +0.000, E1  +383.347, E3 -470397.627}
SPL {X  -159.990, Y  +659.180, Z    +0.000, E1  +383.314, E3 -470411.475}
SPL {X  -159.990, Y  +661.392, Z    +0.000, E1  +383.318, E3 -470422.369}
SPL {X  -159.990, Y  +663.662, Z    +0.000, E1  +383.322, E3 -470433.493}
SPL {X  -159.990, Y  +665.964, Z    +0.000, E1  +383.328, E3 -470444.783}
SPL {X  -159.990, Y  +668.989, Z    +0.000, E1  +383.359, E3 -470459.619}
SPL {X  -159.990, Y  +671.893, Z    +0.000, E1  +383.319, E3 -470473.999}
SPL {X  -159.974, Y  +673.789, Z    +0.000, E1  +383.323, E3 -470483.315}
SPL {X  -159.924, Y  +676.110, Z    +0.000, E1  +383.320, E3 -470494.800}
SPL {X  -159.801, Y  +679.265, Z    +0.000, E1  +383.327, E3 -470510.418}
SPL {X  -159.626, Y  +682.287, Z    +0.000, E1  +383.280, E3 -470525.517}
SPL {X  -159.462, Y  +684.486, Z    +0.000, E1  +383.258, E3 -470536.516}
SPL {X  -159.212, Y  +687.262, Z    +0.000, E1  +383.238, E3 -470550.420}
SPL {X  -158.971, Y  +689.529, Z    +0.000, E1  +383.181, E3 -470561.880}
SPL {X  -158.658, Y  +692.098, Z    +0.000, E1  +383.176, E3 -470574.786}
ENDSPLINE

SPLINE
SPL {X  -159.063, Y  +688.696, Z    +0.000, E1  +377.094, E3 -470617.005}
SPL {X  -159.987, Y  +672.488, Z    +0.000, E1  +365.638, E3 -470641.070}
SPL {X  -159.990, Y  +663.928, Z    +0.000, E1  +359.662, E3 -470646.864}
SPL {X  -159.990, Y  +658.009, Z    +0.000, E1  +355.226, E3 -470650.564}
SPL {X  -159.990, Y  +651.879, Z    +0.000, E1  +350.548, E3 -470655.627}
SPL {X  -159.990, Y  +639.151, Z    +0.000, E1  +342.343, E3 -470670.862}
SPL {X  -159.990, Y  +635.956, Z    +0.000, E1  +340.738, E3 -470676.547}
SPL {X  -159.990, Y  +626.634, Z    +0.000, E1  +337.968, E3 -470704.071}
SPL {X  -159.990, Y  +624.622, Z    +0.000, E1  +337.980, E3 -470714.655}
SPL {X  -159.990, Y  +622.489, Z    +0.000, E1  +337.969, E3 -470725.821}
SPL {X  -159.990, Y  +619.267, Z    +0.000, E1  +337.938, E3 -470742.655}
SPL {X  -159.990, Y  +615.467, Z    +0.000, E1  +337.940, E3 -470762.592}
SPL {X  -159.990, Y  +612.600, Z    +0.000, E1  +337.975, E3 -470777.702}
SPL {X  -159.990, Y  +610.646, Z    +0.000, E1  +337.979, E3 -470787.960}
SPL {X  -159.990, Y  +608.810, Z    +0.000, E1  +337.977, E3 -470797.592}
SPL {X  -159.990, Y  +606.481, Z    +0.000, E1  +337.967, E3 -470809.768}
SPL {X  -159.990, Y  +603.419, Z    +0.000, E1  +337.936, E3 -470825.707}
SPL {X  -159.990, Y  +600.642, Z    +0.000, E1  +337.968, E3 -470840.337}
SPL {X  -159.990, Y  +598.568, Z    +0.000, E1  +337.954, E3 -470851.130}
SPL {X  -159.990, Y  +595.493, Z    +0.000, E1  +337.930, E3 -470867.213}
SPL {X  -159.990, Y  +592.865, Z    +0.000, E1  +337.964, E3 -470881.042}
SPL {X  -159.990, Y  +590.803, Z    +0.000, E1  +337.954, E3 -470891.832}
SPL {X  -159.990, Y  +588.288, Z    +0.000, E1  +337.950, E3 -470904.996}
SPL {X  -159.990, Y  +586.040, Z    +0.000, E1  +337.954, E3 -470916.741}
SPL {X  -159.990, Y  +584.080, Z    +0.000, E1  +337.953, E3 -470927.002}
SPL {X  -159.990, Y  +581.924, Z    +0.000, E1  +337.949, E3 -470938.302}
SPL {X  -159.990, Y  +579.673, Z    +0.000, E1  +337.950, E3 -470950.100}
SPL {X  -159.990, Y  +576.961, Z    +0.000, E1  +337.936, E3 -470964.280}
SPL {X  -159.990, Y  +574.188, Z    +0.000, E1  +337.947, E3 -470978.827}
SPL {X  -159.990, Y  +571.954, Z    +0.000, E1  +337.959, E3 -470990.584}
SPL {X  -159.990, Y  +570.110, Z    +0.000, E1  +337.958, E3 -471000.235}
SPL {X  -159.990, Y  +568.165, Z    +0.000, E1  +337.957, E3 -471010.415}
SPL {X  -159.990, Y  +566.106, Z    +0.000, E1  +337.954, E3 -471021.198}
SPL {X  -159.990, Y  +563.259, Z    +0.000, E1  +337.929, E3 -471036.080}
SPL {X  -159.990, Y  +559.661, Z    +0.000, E1  +337.922, E3 -471054.902}
SPL {X  -159.990, Y  +555.965, Z    +0.000, E1  +337.915, E3 -471074.211}
SPL {X  -159.990, Y  +553.115, Z    +0.000, E1  +337.946, E3 -471089.197}
SPL {X  -159.990, Y  +550.886, Z    +0.000, E1  +337.944, E3 -471100.878}
SPL {X  -159.990, Y  +548.568, Z    +0.000, E1  +337.944, E3 -471112.999}
SPL {X  -159.990, Y  +546.537, Z    +0.000, E1  +337.948, E3 -471123.634}
SPL {X  -159.990, Y  +545.062, Z    +0.000, E1  +337.955, E3 -471131.393}
SPL {X  -159.990, Y  +543.060, Z    +0.000, E1  +337.943, E3 -471141.873}
SPL {X  -159.990, Y  +539.928, Z    +0.000, E1  +337.917, E3 -471158.214}
SPL {X  -159.990, Y  +536.935, Z    +0.000, E1  +337.942, E3 -471173.931}
SPL {X  -159.990, Y  +534.656, Z    +0.000, E1  +337.946, E3 -471185.874}
SPL {X  -159.990, Y  +532.453, Z    +0.000, E1  +337.944, E3 -471197.402}
SPL {X  -159.990, Y  +530.660, Z    +0.000, E1  +337.952, E3 -471206.804}
SPL {X  -159.990, Y  +528.702, Z    +0.000, E1  +337.939, E3 -471217.017}
SPL {X  -159.990, Y  +525.760, Z    +0.000, E1  +337.914, E3 -471232.359}
SPL {X  -159.990, Y  +522.838, Z    +0.000, E1  +337.933, E3 -471247.725}
SPL {X  -159.990, Y  +520.708, Z    +0.000, E1  +337.953, E3 -471258.918}
SPL {X  -159.990, Y  +518.216, Z    +0.000, E1  +337.909, E3 -471271.836}
SPL {X  -159.990, Y  +515.568, Z    +0.000, E1  +338.084, E3 -471287.065}
ENDSPLINE

SPLINE
SPL {X  -159.990, Y  +518.374, Z    +0.000, E1  +341.240, E3 -471299.653}
ENDSPLINE

SPLINE
SPL {X  -159.990, Y  +513.606, Z    +0.000, E1  +339.879, E3 -471315.563}
SPL {X  -159.990, Y  +508.660, Z    +0.000, E1  +338.515, E3 -471330.993}
SPL {X  -159.990, Y  +505.237, Z    +0.000, E1  +337.606, E3 -471341.250}
SPL {X  -159.990, Y  +501.963, Z    +0.000, E1  +336.712, E3 -471350.354}
SPL {X  -159.990, Y  +498.406, Z    +0.000, E1  +335.789, E3 -471360.105}
SPL {X  -159.990, Y  +494.693, Z    +0.000, E1  +334.929, E3 -471370.572}
SPL {X  -159.990, Y  +491.649, Z    +0.000, E1  +334.596, E3 -471381.775}
SPL {X  -159.990, Y  +488.807, Z    +0.000, E1  +334.603, E3 -471394.499}
SPL {X  -159.990, Y  +486.070, Z    +0.000, E1  +334.601, E3 -471406.730}
SPL {X  -159.990, Y  +483.747, Z    +0.000, E1  +334.616, E3 -471417.143}
SPL {X  -159.990, Y  +481.038, Z    +0.000, E1  +334.588, E3 -471429.198}
SPL {X  -159.990, Y  +477.508, Z    +0.000, E1  +334.590, E3 -471444.981}
SPL {X  -159.990, Y  +473.634, Z    +0.000, E1  +334.574, E3 -471462.270}
SPL {X  -159.990, Y  +470.047, Z    +0.000, E1  +334.598, E3 -471478.351}
SPL {X  -159.990, Y  +467.082, Z    +0.000, E1  +334.601, E3 -471491.598}
SPL {X  -159.990, Y  +464.063, Z    +0.000, E1  +334.595, E3 -471505.093}
SPL {X  -159.990, Y  +460.712, Z    +0.000, E1  +334.589, E3 -471520.052}
SPL {X  -159.990, Y  +457.497, Z    +0.000, E1  +334.597, E3 -471534.425}
SPL {X  -159.990, Y  +454.323, Z    +0.000, E1  +334.588, E3 -471548.584}
SPL {X  -159.990, Y  +450.823, Z    +0.000, E1  +334.583, E3 -471564.213}
SPL {X  -159.990, Y  +447.982, Z    +0.000, E1  +334.607, E3 -471576.953}
SPL {X  -159.990, Y  +445.108, Z    +0.000, E1  +334.593, E3 -471589.830}
SPL {X  -159.990, Y  +441.797, Z    +0.000, E1  +334.610, E3 -471604.709}
SPL {X  -159.990, Y  +439.442, Z    +0.000, E1  +334.631, E3 -471615.287}
SPL {X  -159.990, Y  +436.316, Z    +0.000, E1  +334.580, E3 -471629.169}
SPL {X  -159.990, Y  +432.613, Z    +0.000, E1  +334.610, E3 -471645.794}
SPL {X  -159.990, Y  +429.827, Z    +0.000, E1  +334.620, E3 -471658.271}
SPL {X  -159.990, Y  +426.865, Z    +0.000, E1  +334.602, E3 -471671.476}
SPL {X  -159.990, Y  +423.417, Z    +0.000, E1  +334.600, E3 -471686.892}
SPL {X  -159.990, Y  +420.283, Z    +0.000, E1  +334.614, E3 -471700.936}
SPL {X  -159.990, Y  +417.103, Z    +0.000, E1  +334.600, E3 -471715.131}
SPL {X  -159.990, Y  +413.684, Z    +0.000, E1  +334.603, E3 -471730.430}
SPL {X  -159.990, Y  +410.645, Z    +0.000, E1  +334.615, E3 -471744.042}
SPL {X  -159.990, Y  +407.450, Z    +0.000, E1  +334.599, E3 -471758.291}
SPL {X  -159.990, Y  +403.513, Z    +0.000, E1  +334.580, E3 -471775.844}
SPL {X  -159.990, Y  +399.294, Z    +0.000, E1  +334.582, E3 -471794.724}
SPL {X  -159.990, Y  +395.411, Z    +0.000, E1  +334.600, E3 -471812.139}
SPL {X  -159.990, Y  +392.473, Z    +0.000, E1  +334.623, E3 -471825.324}
SPL {X  -159.990, Y  +390.187, Z    +0.000, E1  +334.622, E3 -471835.582}
SPL {X  -159.990, Y  +387.503, Z    +0.000, E1  +334.622, E3 -471847.577}
SPL {X  -159.990, Y  +384.711, Z    +0.000, E1  +334.612, E3 -471860.020}
SPL {X  -159.988, Y  +381.794, Z    +0.000, E1  +334.611, E3 -471873.055}
SPL {X  -159.958, Y  +379.279, Z    +0.000, E1  +334.625, E3 -471884.346}
SPL {X  -159.867, Y  +376.223, Z    +0.000, E1  +334.608, E3 -471898.060}
SPL {X  -159.727, Y  +373.325, Z    +0.000, E1  +334.659, E3 -471911.225}
SPL {X  -159.549, Y  +370.634, Z    +0.000, E1  +334.653, E3 -471923.398}
SPL {X  -159.201, Y  +366.633, Z    +0.000, E1  +334.686, E3 -471941.590}
SPL {X  -158.798, Y  +363.007, Z    +0.000, E1  +334.761, E3 -471958.248}
SPL {X  -158.453, Y  +360.380, Z    +0.000, E1  +334.828, E3 -471970.392}
SPL {X  -158.127, Y  +358.155, Z    +0.000, E1  +334.874, E3 -471980.723}
SPL {X  -158.095, Y  +357.947, Z    +0.000, E1  +338.259, E3 -472012.295}
ENDSPLINE

SPLINE
SPL {X  -158.454, Y  +360.384, Z    +0.000, E1  +340.634, E3 -472024.447}
SPL {X  -159.737, Y  +373.507, Z    +0.000, E1  +349.689, E3 -472046.482}
SPL {X  -159.990, Y  +382.574, Z    +0.000, E1  +355.537, E3 -472053.170}
SPL {X  -159.990, Y  +387.496, Z    +0.000, E1  +358.996, E3 -472055.915}
SPL {X  -159.990, Y  +395.121, Z    +0.000, E1  +364.514, E3 -472060.227}
SPL {X  -159.990, Y  +407.941, Z    +0.000, E1  +374.126, E3 -472072.301}
SPL {X  -159.990, Y  +418.671, Z    +0.000, E1  +379.855, E3 -472091.718}
SPL {X  -159.990, Y  +428.534, Z    +0.000, E1  +383.299, E3 -472115.238}
SPL {X  -159.990, Y  +430.313, Z    +0.000, E1  +383.313, E3 -472123.951}
SPL {X  -159.990, Y  +432.766, Z    +0.000, E1  +383.321, E3 -472135.995}
SPL {X  -159.990, Y  +434.794, Z    +0.000, E1  +383.304, E3 -472146.026}
SPL {X  -159.990, Y  +437.007, Z    +0.000, E1  +383.323, E3 -472156.879}
SPL {X  -159.990, Y  +439.778, Z    +0.000, E1  +383.323, E3 -472170.511}
SPL {X  -159.990, Y  +442.010, Z    +0.000, E1  +383.308, E3 -472181.532}
SPL {X  -159.990, Y  +443.729, Z    +0.000, E1  +383.310, E3 -472189.989}
SPL {X  -159.990, Y  +446.037, Z    +0.000, E1  +383.324, E3 -472201.326}
SPL {X  -159.990, Y  +448.341, Z    +0.000, E1  +383.317, E3 -472212.643}
SPL {X  -159.990, Y  +450.345, Z    +0.000, E1  +383.316, E3 -472222.521}
SPL {X  -159.990, Y  +452.828, Z    +0.000, E1  +383.330, E3 -472234.720}
SPL {X  -159.990, Y  +455.244, Z    +0.000, E1  +383.317, E3 -472246.620}
SPL {X  -159.990, Y  +457.167, Z    +0.000, E1  +383.324, E3 -472256.051}
SPL {X  -159.990, Y  +459.480, Z    +0.000, E1  +383.323, E3 -472267.454}
SPL {X  -159.990, Y  +462.520, Z    +0.000, E1  +383.350, E3 -472282.358}
SPL {X  -159.990, Y  +465.602, Z    +0.000, E1  +383.328, E3 -472297.558}
SPL {X  -159.990, Y  +467.934, Z    +0.000, E1  +383.321, E3 -472309.052}
SPL {X  -159.990, Y  +469.939, Z    +0.000, E1  +383.319, E3 -472318.914}
SPL {X  -159.990, Y  +472.144, Z    +0.000, E1  +383.327, E3 -472329.765}
SPL {X  -159.990, Y  +474.994, Z    +0.000, E1  +383.334, E3 -472343.813}
SPL {X  -159.990, Y  +477.323, Z    +0.000, E1  +383.307, E3 -472355.328}
SPL {X  -159.990, Y  +479.553, Z    +0.000, E1  +383.328, E3 -472366.264}
SPL {X  -159.990, Y  +482.799, Z    +0.000, E1  +383.343, E3 -472382.203}
SPL {X  -159.990, Y  +485.299, Z    +0.000, E1  +383.310, E3 -472394.588}
SPL {X  -159.990, Y  +487.362, Z    +0.000, E1  +383.320, E3 -472404.721}
SPL {X  -159.990, Y  +490.503, Z    +0.000, E1  +383.351, E3 -472420.117}
SPL {X  -159.990, Y  +493.610, Z    +0.000, E1  +383.323, E3 -472435.465}
SPL {X  -159.990, Y  +495.794, Z    +0.000, E1  +383.312, E3 -472446.239}
SPL {X  -159.990, Y  +497.668, Z    +0.000, E1  +383.317, E3 -472455.448}
SPL {X  -159.990, Y  +499.995, Z    +0.000, E1  +383.324, E3 -472466.886}
SPL {X  -159.990, Y  +502.341, Z    +0.000, E1  +383.320, E3 -472478.445}
SPL {X  -159.990, Y  +504.419, Z    +0.000, E1  +383.313, E3 -472488.687}
SPL {X  -159.990, Y  +507.187, Z    +0.000, E1  +383.346, E3 -472502.240}
SPL {X  -159.990, Y  +510.344, Z    +0.000, E1  +383.327, E3 -472517.825}
SPL {X  -159.990, Y  +512.484, Z    +0.000, E1  +383.309, E3 -472528.398}
SPL {X  -159.990, Y  +514.016, Z    +0.000, E1  +383.308, E3 -472535.946}
SPL {X  -159.990, Y  +516.195, Z    +0.000, E1  +383.325, E3 -472546.634}
SPL {X  -159.990, Y  +518.925, Z    +0.000, E1  +383.333, E3 -472559.997}
SPL {X  -159.990, Y  +521.408, Z    +0.000, E1  +383.329, E3 -472572.206}
SPL {X  -159.990, Y  +523.942, Z    +0.000, E1  +383.333, E3 -472584.699}
SPL {X  -159.990, Y  +527.007, Z    +0.000, E1  +383.339, E3 -472599.799}
SPL {X  -159.990, Y  +529.993, Z    +0.000, E1  +383.329, E3 -472614.501}
SPL {X  -159.990, Y  +532.441, Z    +0.000, E1  +383.322, E3 -472626.552}
SPL {X  -159.990, Y  +534.618, Z    +0.000, E1  +383.322, E3 -472637.285}
SPL {X  -159.990, Y  +537.024, Z    +0.000, E1  +383.321, E3 -472649.147}
SPL {X  -159.990, Y  +539.129, Z    +0.000, E1  +383.310, E3 -472659.530}
SPL {X  -159.990, Y  +541.183, Z    +0.000, E1  +383.319, E3 -472669.627}
SPL {X  -159.990, Y  +543.647, Z    +0.000, E1  +383.325, E3 -472681.730}
SPL {X  -159.990, Y  +546.832, Z    +0.000, E1  +383.349, E3 -472697.353}
SPL {X  -159.990, Y  +549.756, Z    +0.000, E1  +383.320, E3 -472711.794}
SPL {X  -159.990, Y  +551.655, Z    +0.000, E1  +383.320, E3 -472721.145}
SPL {X  -159.990, Y  +553.711, Z    +0.000, E1  +383.317, E3 -472731.267}
SPL {X  -159.990, Y  +555.637, Z    +0.000, E1  +383.323, E3 -472740.735}
SPL {X  -159.990, Y  +558.758, Z    +0.000, E1  +383.351, E3 -472756.045}
SPL {X  -159.990, Y  +561.830, Z    +0.000, E1  +383.325, E3 -472771.218}
SPL {X  -159.990, Y  +564.273, Z    +0.000, E1  +383.325, E3 -472783.243}
SPL {X  -159.990, Y  +567.351, Z    +0.000, E1  +383.348, E3 -472798.338}
SPL {X  -159.990, Y  +570.314, Z    +0.000, E1  +383.326, E3 -472812.970}
SPL {X  -159.990, Y  +572.504, Z    +0.000, E1  +383.321, E3 -472823.755}
SPL {X  -159.990, Y  +575.653, Z    +0.000, E1  +383.355, E3 -472839.192}
SPL {X  -159.990, Y  +578.932, Z    +0.000, E1  +383.330, E3 -472855.375}
SPL {X  -159.990, Y  +581.497, Z    +0.000, E1  +383.329, E3 -472867.959}
SPL {X  -159.990, Y  +583.973, Z    +0.000, E1  +383.332, E3 -472880.145}
SPL {X  -159.990, Y  +586.877, Z    +0.000, E1  +383.349, E3 -472894.399}
SPL {X  -159.990, Y  +590.594, Z    +0.000, E1  +383.363, E3 -472912.649}
SPL {X  -159.990, Y  +593.847, Z    +0.000, E1  +383.340, E3 -472928.660}
SPL {X  -159.990, Y  +596.027, Z    +0.000, E1  +383.330, E3 -472939.406}
SPL {X  -159.990, Y  +599.017, Z    +0.000, E1  +383.373, E3 -472953.971}
SPL {X  -159.990, Y  +601.949, Z    +0.000, E1  +383.344, E3 -472968.423}
SPL {X  -159.990, Y  +604.315, Z    +0.000, E1  +383.350, E3 -472980.048}
SPL {X  -159.990, Y  +607.388, Z    +0.000, E1  +383.369, E3 -472995.113}
SPL {X  -159.990, Y  +610.073, Z    +0.000, E1  +383.343, E3 -473008.378}
SPL {X  -159.990, Y  +612.330, Z    +0.000, E1  +383.340, E3 -473019.505}
SPL {X  -159.990, Y  +615.036, Z    +0.000, E1  +383.353, E3 -473032.792}
SPL {X  -159.990, Y  +618.481, Z    +0.000, E1  +383.366, E3 -473049.731}
SPL {X  -159.990, Y  +621.517, Z    +0.000, E1  +383.337, E3 -473064.713}
SPL {X  -159.990, Y  +623.764, Z    +0.000, E1  +383.335, E3 -473075.764}
SPL {X  -159.990, Y  +626.608, Z    +0.000, E1  +383.361, E3 -473089.689}
SPL {X  -159.990, Y  +630.271, Z    +0.000, E1  +383.375, E3 -473107.650}
SPL {X  -159.990, Y  +633.318, Z    +0.000, E1  +383.339, E3 -473122.728}
SPL {X  -159.990, Y  +635.650, Z    +0.000, E1  +383.339, E3 -473134.198}
SPL {X  -159.990, Y  +638.406, Z    +0.000, E1  +383.354, E3 -473147.765}
SPL {X  -159.990, Y  +641.831, Z    +0.000, E1  +383.342, E3 -473164.713}
SPL {X  -159.990, Y  +644.884, Z    +0.000, E1  +383.324, E3 -473179.799}
SPL {X  -159.990, Y  +647.550, Z    +0.000, E1  +383.318, E3 -473192.966}
SPL {X  -159.990, Y  +650.790, Z    +0.000, E1  +383.346, E3 -473208.833}
SPL {X  -159.990, Y  +654.543, Z    +0.000, E1  +383.348, E3 -473227.286}
SPL {X  -159.990, Y  +658.319, Z    +0.000, E1  +383.349, E3 -473245.875}
SPL {X  -159.990, Y  +661.392, Z    +0.000, E1  +383.318, E3 -473261.078}
SPL {X  -159.990, Y  +663.662, Z    +0.000, E1  +383.322, E3 -473272.202}
SPL {X  -159.990, Y  +665.964, Z    +0.000, E1  +383.328, E3 -473283.493}
SPL {X  -159.990, Y  +667.870, Z    +0.000, E1  +383.320, E3 -473292.900}
SPL {X  -159.990, Y  +669.861, Z    +0.000, E1  +383.321, E3 -473302.701}
SPL {X  -159.990, Y  +671.893, Z    +0.000, E1  +383.319, E3 -473312.709}
SPL {X  -159.974, Y  +673.789, Z    +0.000, E1  +383.323, E3 -473322.025}
SPL {X  -159.924, Y  +676.110, Z    +0.000, E1  +383.320, E3 -473333.509}
SPL {X  -159.801, Y  +679.265, Z    +0.000, E1  +383.327, E3 -473349.128}
SPL {X  -159.626, Y  +682.287, Z    +0.000, E1  +383.280, E3 -473364.226}
SPL {X  -159.462, Y  +684.486, Z    +0.000, E1  +383.258, E3 -473375.226}
SPL {X  -159.212, Y  +687.262, Z    +0.000, E1  +383.238, E3 -473389.130}
SPL {X  -158.861, Y  +690.475, Z    +0.000, E1  +383.199, E3 -473405.298}
SPL {X  -158.553, Y  +692.896, Z    +0.000, E1  +383.130, E3 -473417.594}
ENDSPLINE

SPLINE
SPL {X  -159.063, Y  +688.696, Z    +0.000, E1  +377.094, E3 -473455.715}
SPL {X  -159.957, Y  +674.769, Z    +0.000, E1  +367.092, E3 -473478.096}
SPL {X  -159.990, Y  +671.516, Z    +0.000, E1  +364.944, E3 -473480.482}
SPL {X  -159.990, Y  +663.928, Z    +0.000, E1  +359.662, E3 -473485.574}
SPL {X  -159.990, Y  +658.009, Z    +0.000, E1  +355.226, E3 -473489.274}
SPL {X  -159.990, Y  +651.879, Z    +0.000, E1  +350.548, E3 -473494.337}
SPL {X  -159.990, Y  +637.832, Z    +0.000, E1  +341.694, E3 -473511.928}
SPL {X  -159.990, Y  +626.634, Z    +0.000, E1  +337.968, E3 -473542.781}
SPL {X  -159.990, Y  +624.622, Z    +0.000, E1  +337.980, E3 -473553.364}
SPL {X  -159.990, Y  +622.489, Z    +0.000, E1  +337.969, E3 -473564.531}
SPL {X  -159.990, Y  +619.955, Z    +0.000, E1  +337.968, E3 -473577.821}
SPL {X  -159.990, Y  +617.386, Z    +0.000, E1  +337.968, E3 -473591.296}
SPL {X  -159.990, Y  +614.863, Z    +0.000, E1  +337.969, E3 -473604.528}
SPL {X  -159.990, Y  +612.600, Z    +0.000, E1  +337.975, E3 -473616.412}
SPL {X  -159.990, Y  +610.646, Z    +0.000, E1  +337.979, E3 -473626.669}
SPL {X  -159.990, Y  +608.810, Z    +0.000, E1  +337.977, E3 -473636.302}
SPL {X  -159.990, Y  +605.804, Z    +0.000, E1  +337.936, E3 -473651.947}
SPL {X  -159.990, Y  +602.819, Z    +0.000, E1  +337.963, E3 -473667.619}
SPL {X  -159.990, Y  +600.642, Z    +0.000, E1  +337.968, E3 -473679.047}
SPL {X  -159.990, Y  +598.568, Z    +0.000, E1  +337.954, E3 -473689.839}
SPL {X  -159.990, Y  +595.493, Z    +0.000, E1  +337.930, E3 -473705.923}
SPL {X  -159.990, Y  +592.865, Z    +0.000, E1  +337.964, E3 -473719.751}
SPL {X  -159.990, Y  +590.803, Z    +0.000, E1  +337.954, E3 -473730.542}
SPL {X  -159.990, Y  +588.288, Z    +0.000, E1  +337.950, E3 -473743.706}
SPL {X  -159.990, Y  +586.040, Z    +0.000, E1  +337.954, E3 -473755.451}
SPL {X  -159.990, Y  +584.080, Z    +0.000, E1  +337.953, E3 -473765.711}
SPL {X  -159.990, Y  +581.924, Z    +0.000, E1  +337.949, E3 -473777.012}
SPL {X  -159.990, Y  +579.673, Z    +0.000, E1  +337.950, E3 -473788.810}
SPL {X  -159.990, Y  +576.961, Z    +0.000, E1  +337.936, E3 -473802.989}
SPL {X  -159.990, Y  +574.188, Z    +0.000, E1  +337.947, E3 -473817.536}
SPL {X  -159.990, Y  +571.954, Z    +0.000, E1  +337.959, E3 -473829.294}
SPL {X  -159.990, Y  +570.110, Z    +0.000, E1  +337.958, E3 -473838.944}
SPL {X  -159.990, Y  +568.165, Z    +0.000, E1  +337.957, E3 -473849.124}
SPL {X  -159.990, Y  +565.292, Z    +0.000, E1  +337.922, E3 -473864.102}
SPL {X  -159.990, Y  +562.598, Z    +0.000, E1  +337.958, E3 -473878.313}
SPL {X  -159.990, Y  +560.652, Z    +0.000, E1  +337.962, E3 -473888.525}
SPL {X  -159.990, Y  +558.143, Z    +0.000, E1  +337.928, E3 -473901.557}
SPL {X  -159.990, Y  +555.329, Z    +0.000, E1  +337.943, E3 -473916.301}
SPL {X  -159.990, Y  +553.115, Z    +0.000, E1  +337.946, E3 -473927.907}
SPL {X  -159.990, Y  +550.886, Z    +0.000, E1  +337.944, E3 -473939.588}
SPL {X  -159.990, Y  +548.568, Z    +0.000, E1  +337.944, E3 -473951.709}
SPL {X  -159.990, Y  +545.859, Z    +0.000, E1  +337.926, E3 -473965.859}
SPL {X  -159.990, Y  +542.390, Z    +0.000, E1  +337.914, E3 -473984.029}
SPL {X  -159.990, Y  +539.341, Z    +0.000, E1  +337.944, E3 -474000.051}
SPL {X  -159.990, Y  +536.935, Z    +0.000, E1  +337.942, E3 -474012.640}
SPL {X  -159.990, Y  +534.656, Z    +0.000, E1  +337.946, E3 -474024.584}
SPL {X  -159.990, Y  +531.679, Z    +0.000, E1  +337.913, E3 -474040.098}
SPL {X  -159.990, Y  +527.941, Z    +0.000, E1  +337.907, E3 -474059.640}
SPL {X  -159.990, Y  +525.053, Z    +0.000, E1  +337.942, E3 -474074.830}
SPL {X  -159.990, Y  +522.838, Z    +0.000, E1  +337.933, E3 -474086.435}
SPL {X  -159.990, Y  +519.698, Z    +0.000, E1  +337.916, E3 -474102.818}
SPL {X  -159.990, Y  +517.251, Z    +0.000, E1  +337.946, E3 -474115.678}
SPL {X  -159.990, Y  +515.568, Z    +0.000, E1  +338.084, E3 -474125.775}
ENDSPLINE

SPLINE
SPL {X  -159.990, Y  +517.293, Z    +0.000, E1  +340.923, E3 -474142.073}
ENDSPLINE

SPLINE
SPL {X  -159.990, Y  +512.548, Z    +0.000, E1  +339.587, E3 -474157.648}
SPL {X  -159.990, Y  +508.660, Z    +0.000, E1  +338.515, E3 -474169.702}
SPL {X  -159.990, Y  +503.499, Z    +0.000, E1  +337.116, E3 -474184.782}
SPL {X  -159.990, Y  +498.406, Z    +0.000, E1  +335.789, E3 -474198.815}
SPL {X  -159.990, Y  +494.693, Z    +0.000, E1  +334.929, E3 -474209.282}
SPL {X  -159.990, Y  +491.649, Z    +0.000, E1  +334.596, E3 -474220.484}
SPL {X  -159.990, Y  +488.807, Z    +0.000, E1  +334.603, E3 -474233.209}
SPL {X  -159.990, Y  +486.070, Z    +0.000, E1  +334.601, E3 -474245.440}
SPL {X  -159.990, Y  +483.747, Z    +0.000, E1  +334.616, E3 -474255.853}
SPL {X  -159.990, Y  +481.038, Z    +0.000, E1  +334.588, E3 -474267.908}
SPL {X  -159.990, Y  +477.508, Z    +0.000, E1  +334.590, E3 -474283.690}
SPL {X  -159.990, Y  +473.634, Z    +0.000, E1  +334.574, E3 -474300.979}
SPL {X  -159.990, Y  +470.047, Z    +0.000, E1  +334.598, E3 -474317.060}
SPL {X  -159.990, Y  +467.082, Z    +0.000, E1  +334.601, E3 -474330.307}
SPL {X  -159.990, Y  +464.063, Z    +0.000, E1  +334.595, E3 -474343.802}
SPL {X  -159.990, Y  +460.712, Z    +0.000, E1  +334.589, E3 -474358.762}
SPL {X  -159.990, Y  +457.497, Z    +0.000, E1  +334.597, E3 -474373.134}
SPL {X  -159.990, Y  +455.126, Z    +0.000, E1  +334.611, E3 -474383.743}
SPL {X  -159.990, Y  +453.438, Z    +0.000, E1  +334.615, E3 -474391.303}
SPL {X  -159.990, Y  +450.823, Z    +0.000, E1  +334.583, E3 -474402.923}
SPL {X  -159.990, Y  +446.894, Z    +0.000, E1  +334.572, E3 -474420.480}
SPL {X  -159.990, Y  +443.345, Z    +0.000, E1  +334.610, E3 -474436.487}
SPL {X  -159.990, Y  +441.077, Z    +0.000, E1  +334.631, E3 -474446.685}
SPL {X  -159.990, Y  +438.608, Z    +0.000, E1  +334.608, E3 -474457.682}
SPL {X  -159.990, Y  +434.852, Z    +0.000, E1  +334.585, E3 -474474.436}
SPL {X  -159.990, Y  +430.645, Z    +0.000, E1  +334.586, E3 -474493.256}
SPL {X  -159.990, Y  +426.865, Z    +0.000, E1  +334.602, E3 -474510.185}
SPL {X  -159.990, Y  +423.417, Z    +0.000, E1  +334.600, E3 -474525.601}
SPL {X  -159.990, Y  +419.467, Z    +0.000, E1  +334.583, E3 -474543.236}
SPL {X  -159.990, Y  +416.355, Z    +0.000, E1  +334.625, E3 -474557.233}
SPL {X  -159.990, Y  +413.684, Z    +0.000, E1  +334.603, E3 -474569.140}
SPL {X  -159.990, Y  +410.645, Z    +0.000, E1  +334.615, E3 -474582.752}
SPL {X  -159.990, Y  +408.351, Z    +0.000, E1  +334.628, E3 -474593.038}
SPL {X  -159.990, Y  +406.574, Z    +0.000, E1  +334.625, E3 -474600.955}
SPL {X  -159.990, Y  +404.255, Z    +0.000, E1  +334.609, E3 -474611.291}
SPL {X  -159.990, Y  +401.103, Z    +0.000, E1  +334.596, E3 -474625.355}
SPL {X  -159.990, Y  +398.389, Z    +0.000, E1  +334.619, E3 -474637.551}
SPL {X  -159.990, Y  +395.411, Z    +0.000, E1  +334.600, E3 -474650.848}
SPL {X  -159.990, Y  +392.473, Z    +0.000, E1  +334.623, E3 -474664.033}
SPL {X  -159.990, Y  +390.187, Z    +0.000, E1  +334.622, E3 -474674.292}
SPL {X  -159.990, Y  +387.503, Z    +0.000, E1  +334.622, E3 -474686.286}
SPL {X  -159.990, Y  +384.711, Z    +0.000, E1  +334.612, E3 -474698.730}
SPL {X  -159.988, Y  +381.794, Z    +0.000, E1  +334.611, E3 -474711.765}
SPL {X  -159.958, Y  +379.279, Z    +0.000, E1  +334.625, E3 -474723.055}
SPL {X  -159.867, Y  +376.223, Z    +0.000, E1  +334.608, E3 -474736.770}
SPL {X  -159.727, Y  +373.325, Z    +0.000, E1  +334.659, E3 -474749.935}
SPL {X  -159.549, Y  +370.634, Z    +0.000, E1  +334.653, E3 -474762.108}
SPL {X  -159.201, Y  +366.633, Z    +0.000, E1  +334.686, E3 -474780.300}
SPL {X  -158.798, Y  +363.007, Z    +0.000, E1  +334.761, E3 -474796.958}
SPL {X  -158.453, Y  +360.380, Z    +0.000, E1  +334.828, E3 -474809.102}
SPL {X  -158.127, Y  +358.155, Z    +0.000, E1  +334.874, E3 -474819.433}
SPL {X  -158.095, Y  +357.947, Z    +0.000, E1  +338.259, E3 -474851.005}
ENDSPLINE

SPLINE
SPL {X  -158.454, Y  +360.384, Z    +0.000, E1  +340.634, E3 -474863.156}
SPL {X  -159.737, Y  +373.507, Z    +0.000, E1  +349.689, E3 -474885.192}
SPL {X  -159.990, Y  +382.574, Z    +0.000, E1  +355.537, E3 -474891.879}
SPL {X  -159.990, Y  +389.909, Z    +0.000, E1  +360.662, E3 -474895.894}
SPL {X  -159.990, Y  +396.289, Z    +0.000, E1  +365.500, E3 -474899.674}
SPL {X  -159.990, Y  +407.941, Z    +0.000, E1  +374.126, E3 -474911.011}
SPL {X  -159.990, Y  +418.671, Z    +0.000, E1  +379.855, E3 -474930.427}
SPL {X  -159.990, Y  +429.878, Z    +0.000, E1  +383.330, E3 -474960.482}
SPL {X  -159.990, Y  +432.766, Z    +0.000, E1  +383.321, E3 -474974.705}
SPL {X  -159.990, Y  +434.794, Z    +0.000, E1  +383.304, E3 -474984.736}
SPL {X  -159.990, Y  +437.007, Z    +0.000, E1  +383.323, E3 -474995.589}
SPL {X  -159.990, Y  +439.778, Z    +0.000, E1  +383.323, E3 -475009.221}
SPL {X  -159.990, Y  +442.010, Z    +0.000, E1  +383.308, E3 -475020.242}
SPL {X  -159.990, Y  +443.729, Z    +0.000, E1  +383.310, E3 -475028.698}
SPL {X  -159.990, Y  +446.037, Z    +0.000, E1  +383.324, E3 -475040.035}
SPL {X  -159.990, Y  +448.341, Z    +0.000, E1  +383.317, E3 -475051.353}
SPL {X  -159.990, Y  +450.345, Z    +0.000, E1  +383.316, E3 -475061.231}
SPL {X  -159.990, Y  +452.828, Z    +0.000, E1  +383.330, E3 -475073.430}
SPL {X  -159.990, Y  +455.244, Z    +0.000, E1  +383.317, E3 -475085.330}
SPL {X  -159.990, Y  +457.167, Z    +0.000, E1  +383.324, E3 -475094.760}
SPL {X  -159.990, Y  +459.480, Z    +0.000, E1  +383.323, E3 -475106.164}
SPL {X  -159.990, Y  +462.520, Z    +0.000, E1  +383.350, E3 -475121.068}
SPL {X  -159.990, Y  +465.602, Z    +0.000, E1  +383.328, E3 -475136.268}
SPL {X  -159.990, Y  +467.934, Z    +0.000, E1  +383.321, E3 -475147.762}
SPL {X  -159.990, Y  +469.939, Z    +0.000, E1  +383.319, E3 -475157.624}
SPL {X  -159.990, Y  +472.144, Z    +0.000, E1  +383.327, E3 -475168.474}
SPL {X  -159.990, Y  +474.994, Z    +0.000, E1  +383.334, E3 -475182.523}
SPL {X  -159.990, Y  +477.323, Z    +0.000, E1  +383.307, E3 -475194.038}
SPL {X  -159.990, Y  +479.553, Z    +0.000, E1  +383.328, E3 -475204.973}
SPL {X  -159.990, Y  +482.799, Z    +0.000, E1  +383.343, E3 -475220.912}
SPL {X  -159.990, Y  +485.299, Z    +0.000, E1  +383.310, E3 -475233.297}
SPL {X  -159.990, Y  +488.031, Z    +0.000, E1  +383.345, E3 -475246.676}
SPL {X  -159.990, Y  +491.121, Z    +0.000, E1  +383.323, E3 -475261.922}
SPL {X  -159.990, Y  +493.610, Z    +0.000, E1  +383.323, E3 -475274.175}
SPL {X  -159.990, Y  +496.863, Z    +0.000, E1  +383.350, E3 -475290.135}
SPL {X  -159.990, Y  +499.995, Z    +0.000, E1  +383.324, E3 -475305.596}
SPL {X  -159.990, Y  +502.341, Z    +0.000, E1  +383.320, E3 -475317.155}
SPL {X  -159.990, Y  +505.377, Z    +0.000, E1  +383.346, E3 -475332.046}
SPL {X  -159.990, Y  +508.697, Z    +0.000, E1  +383.335, E3 -475348.405}
SPL {X  -159.990, Y  +511.771, Z    +0.000, E1  +383.331, E3 -475363.552}
SPL {X  -159.990, Y  +514.016, Z    +0.000, E1  +383.308, E3 -475374.656}
SPL {X  -159.990, Y  +516.195, Z    +0.000, E1  +383.325, E3 -475385.344}
SPL {X  -159.990, Y  +518.925, Z    +0.000, E1  +383.333, E3 -475398.707}
SPL {X  -159.990, Y  +521.408, Z    +0.000, E1  +383.329, E3 -475410.916}
SPL {X  -159.990, Y  +523.942, Z    +0.000, E1  +383.333, E3 -475423.409}
SPL {X  -159.990, Y  +526.221, Z    +0.000, E1  +383.314, E3 -475434.685}
SPL {X  -159.990, Y  +527.834, Z    +0.000, E1  +383.311, E3 -475442.635}
SPL {X  -159.990, Y  +529.993, Z    +0.000, E1  +383.329, E3 -475453.211}
SPL {X  -159.990, Y  +532.441, Z    +0.000, E1  +383.322, E3 -475465.262}
SPL {X  -159.990, Y  +534.618, Z    +0.000, E1  +383.322, E3 -475475.995}
SPL {X  -159.990, Y  +537.024, Z    +0.000, E1  +383.321, E3 -475487.857}
SPL {X  -159.990, Y  +539.129, Z    +0.000, E1  +383.310, E3 -475498.240}
SPL {X  -159.990, Y  +541.183, Z    +0.000, E1  +383.319, E3 -475508.337}
SPL {X  -159.990, Y  +543.647, Z    +0.000, E1  +383.325, E3 -475520.440}
SPL {X  -159.990, Y  +546.832, Z    +0.000, E1  +383.349, E3 -475536.063}
SPL {X  -159.990, Y  +549.756, Z    +0.000, E1  +383.320, E3 -475550.503}
SPL {X  -159.990, Y  +551.655, Z    +0.000, E1  +383.320, E3 -475559.854}
SPL {X  -159.990, Y  +553.711, Z    +0.000, E1  +383.317, E3 -475569.976}
SPL {X  -159.990, Y  +555.637, Z    +0.000, E1  +383.323, E3 -475579.445}
SPL {X  -159.990, Y  +558.758, Z    +0.000, E1  +383.351, E3 -475594.755}
SPL {X  -159.990, Y  +561.830, Z    +0.000, E1  +383.325, E3 -475609.928}
SPL {X  -159.990, Y  +564.273, Z    +0.000, E1  +383.325, E3 -475621.952}
SPL {X  -159.990, Y  +567.351, Z    +0.000, E1  +383.348, E3 -475637.048}
SPL {X  -159.990, Y  +570.314, Z    +0.000, E1  +383.326, E3 -475651.680}
SPL {X  -159.990, Y  +572.504, Z    +0.000, E1  +383.321, E3 -475662.465}
SPL {X  -159.990, Y  +575.653, Z    +0.000, E1  +383.355, E3 -475677.902}
SPL {X  -159.990, Y  +578.932, Z    +0.000, E1  +383.330, E3 -475694.084}
SPL {X  -159.990, Y  +581.497, Z    +0.000, E1  +383.329, E3 -475706.669}
SPL {X  -159.990, Y  +583.973, Z    +0.000, E1  +383.332, E3 -475718.854}
SPL {X  -159.990, Y  +586.020, Z    +0.000, E1  +383.323, E3 -475728.938}
SPL {X  -159.990, Y  +587.711, Z    +0.000, E1  +383.318, E3 -475737.278}
SPL {X  -159.990, Y  +589.763, Z    +0.000, E1  +383.328, E3 -475747.354}
SPL {X  -159.990, Y  +591.698, Z    +0.000, E1  +383.324, E3 -475756.839}
SPL {X  -159.990, Y  +593.847, Z    +0.000, E1  +383.340, E3 -475767.369}
SPL {X  -159.990, Y  +597.018, Z    +0.000, E1  +383.367, E3 -475782.901}
SPL {X  -159.990, Y  +599.887, Z    +0.000, E1  +383.341, E3 -475797.006}
SPL {X  -159.990, Y  +601.949, Z    +0.000, E1  +383.344, E3 -475807.132}
SPL {X  -159.990, Y  +605.106, Z    +0.000, E1  +383.383, E3 -475822.578}
SPL {X  -159.990, Y  +608.111, Z    +0.000, E1  +383.342, E3 -475837.429}
SPL {X  -159.990, Y  +610.073, Z    +0.000, E1  +383.343, E3 -475847.087}
SPL {X  -159.990, Y  +613.021, Z    +0.000, E1  +383.365, E3 -475861.558}
SPL {X  -159.990, Y  +615.657, Z    +0.000, E1  +383.331, E3 -475874.606}
SPL {X  -159.990, Y  +617.658, Z    +0.000, E1  +383.335, E3 -475884.448}
SPL {X  -159.990, Y  +620.788, Z    +0.000, E1  +383.368, E3 -475899.781}
SPL {X  -159.990, Y  +624.347, Z    +0.000, E1  +383.355, E3 -475917.302}
SPL {X  -159.990, Y  +627.144, Z    +0.000, E1  +383.340, E3 -475931.071}
SPL {X  -159.990, Y  +630.271, Z    +0.000, E1  +383.375, E3 -475946.360}
SPL {X  -159.990, Y  +633.318, Z    +0.000, E1  +383.339, E3 -475961.437}
SPL {X  -159.990, Y  +635.650, Z    +0.000, E1  +383.339, E3 -475972.908}
SPL {X  -159.990, Y  +638.406, Z    +0.000, E1  +383.354, E3 -475986.475}
SPL {X  -159.990, Y  +641.831, Z    +0.000, E1  +383.342, E3 -476003.422}
SPL {X  -159.990, Y  +644.884, Z    +0.000, E1  +383.324, E3 -476018.509}
SPL {X  -159.990, Y  +647.550, Z    +0.000, E1  +383.318, E3 -476031.676}
SPL {X  -159.990, Y  +650.790, Z    +0.000, E1  +383.346, E3 -476047.542}
SPL {X  -159.990, Y  +654.543, Z    +0.000, E1  +383.348, E3 -476065.995}
SPL {X  -159.990, Y  +658.319, Z    +0.000, E1  +383.349, E3 -476084.585}
SPL {X  -159.990, Y  +661.392, Z    +0.000, E1  +383.318, E3 -476099.788}
SPL {X  -159.990, Y  +663.662, Z    +0.000, E1  +383.322, E3 -476110.912}
SPL {X  -159.990, Y  +665.964, Z    +0.000, E1  +383.328, E3 -476122.203}
SPL {X  -159.990, Y  +667.870, Z    +0.000, E1  +383.320, E3 -476131.609}
SPL {X  -159.990, Y  +669.861, Z    +0.000, E1  +383.321, E3 -476141.411}
SPL {X  -159.983, Y  +672.946, Z    +0.000, E1  +383.359, E3 -476156.520}
SPL {X  -159.924, Y  +676.110, Z    +0.000, E1  +383.320, E3 -476172.219}
SPL {X  -159.845, Y  +678.302, Z    +0.000, E1  +383.298, E3 -476183.121}
SPL {X  -159.760, Y  +680.081, Z    +0.000, E1  +383.288, E3 -476191.964}
SPL {X  -159.626, Y  +682.287, Z    +0.000, E1  +383.280, E3 -476202.936}
SPL {X  -159.462, Y  +684.486, Z    +0.000, E1  +383.258, E3 -476213.936}
SPL {X  -159.289, Y  +686.457, Z    +0.000, E1  +383.223, E3 -476223.846}
SPL {X  -159.052, Y  +688.801, Z    +0.000, E1  +383.217, E3 -476235.580}
SPL {X  -158.770, Y  +691.222, Z    +0.000, E1  +383.158, E3 -476247.838}
SPL {X  -158.553, Y  +692.896, Z    +0.000, E1  +383.130, E3 -476256.303}
ENDSPLINE

SPLINE
SPL {X  -159.063, Y  +688.696, Z    +0.000, E1  +377.094, E3 -476294.424}
SPL {X  -159.987, Y  +672.488, Z    +0.000, E1  +365.638, E3 -476318.489}
SPL {X  -159.990, Y  +663.928, Z    +0.000, E1  +359.662, E3 -476324.284}
SPL {X  -159.990, Y  +658.009, Z    +0.000, E1  +355.226, E3 -476327.984}
SPL {X  -159.990, Y  +651.879, Z    +0.000, E1  +350.548, E3 -476333.046}
SPL {X  -159.990, Y  +637.832, Z    +0.000, E1  +341.694, E3 -476350.637}
SPL {X  -159.990, Y  +626.634, Z    +0.000, E1  +337.968, E3 -476381.490}
SPL {X  -159.990, Y  +624.622, Z    +0.000, E1  +337.980, E3 -476392.074}
SPL {X  -159.990, Y  +622.489, Z    +0.000, E1  +337.969, E3 -476403.240}
SPL {X  -159.990, Y  +619.955, Z    +0.000, E1  +337.968, E3 -476416.530}
SPL {X  -159.990, Y  +617.386, Z    +0.000, E1  +337.968, E3 -476430.005}
SPL {X  -159.990, Y  +614.863, Z    +0.000, E1  +337.969, E3 -476443.237}
SPL {X  -159.990, Y  +612.600, Z    +0.000, E1  +337.975, E3 -476455.122}
SPL {X  -159.990, Y  +610.646, Z    +0.000, E1  +337.979, E3 -476465.379}
SPL {X  -159.990, Y  +608.810, Z    +0.000, E1  +337.977, E3 -476475.012}
SPL {X  -159.990, Y  +606.481, Z    +0.000, E1  +337.967, E3 -476487.187}
SPL {X  -159.990, Y  +603.419, Z    +0.000, E1  +337.936, E3 -476503.127}
SPL {X  -159.990, Y  +600.642, Z    +0.000, E1  +337.968, E3 -476517.756}
SPL {X  -159.990, Y  +598.568, Z    +0.000, E1  +337.954, E3 -476528.549}
SPL {X  -159.990, Y  +595.493, Z    +0.000, E1  +337.930, E3 -476544.632}
SPL {X  -159.990, Y  +592.865, Z    +0.000, E1  +337.964, E3 -476558.461}
SPL {X  -159.990, Y  +590.803, Z    +0.000, E1  +337.954, E3 -476569.252}
SPL {X  -159.990, Y  +588.288, Z    +0.000, E1  +337.950, E3 -476582.416}
SPL {X  -159.990, Y  +586.040, Z    +0.000, E1  +337.954, E3 -476594.161}
SPL {X  -159.990, Y  +584.080, Z    +0.000, E1  +337.953, E3 -476604.421}
SPL {X  -159.990, Y  +581.924, Z    +0.000, E1  +337.949, E3 -476615.721}
SPL {X  -159.990, Y  +578.886, Z    +0.000, E1  +337.918, E3 -476631.575}
SPL {X  -159.990, Y  +576.252, Z    +0.000, E1  +337.962, E3 -476645.473}
SPL {X  -159.990, Y  +574.188, Z    +0.000, E1  +337.947, E3 -476656.246}
SPL {X  -159.990, Y  +571.954, Z    +0.000, E1  +337.959, E3 -476668.004}
SPL {X  -159.990, Y  +570.110, Z    +0.000, E1  +337.958, E3 -476677.654}
SPL {X  -159.990, Y  +568.165, Z    +0.000, E1  +337.957, E3 -476687.834}
SPL {X  -159.990, Y  +566.106, Z    +0.000, E1  +337.954, E3 -476698.617}
SPL {X  -159.990, Y  +563.259, Z    +0.000, E1  +337.929, E3 -476713.499}
SPL {X  -159.990, Y  +559.661, Z    +0.000, E1  +337.922, E3 -476732.322}
SPL {X  -159.990, Y  +555.965, Z    +0.000, E1  +337.915, E3 -476751.631}
SPL {X  -159.990, Y  +553.115, Z    +0.000, E1  +337.946, E3 -476766.616}
SPL {X  -159.990, Y  +550.886, Z    +0.000, E1  +337.944, E3 -476778.298}
SPL {X  -159.990, Y  +548.568, Z    +0.000, E1  +337.944, E3 -476790.419}
SPL {X  -159.990, Y  +545.859, Z    +0.000, E1  +337.926, E3 -476804.568}
SPL {X  -159.990, Y  +543.060, Z    +0.000, E1  +337.943, E3 -476819.292}
SPL {X  -159.990, Y  +539.928, Z    +0.000, E1  +337.917, E3 -476835.633}
SPL {X  -159.990, Y  +536.935, Z    +0.000, E1  +337.942, E3 -476851.350}
SPL {X  -159.990, Y  +534.656, Z    +0.000, E1  +337.946, E3 -476863.294}
SPL {X  -159.990, Y  +531.679, Z    +0.000, E1  +337.913, E3 -476878.808}
SPL {X  -159.990, Y  +527.941, Z    +0.000, E1  +337.907, E3 -476898.350}
SPL {X  -159.990, Y  +525.053, Z    +0.000, E1  +337.942, E3 -476913.540}
SPL {X  -159.990, Y  +522.838, Z    +0.000, E1  +337.933, E3 -476925.144}
SPL {X  -159.990, Y  +519.698, Z    +0.000, E1  +337.916, E3 -476941.527}
SPL {X  -159.990, Y  +517.251, Z    +0.000, E1  +337.946, E3 -476954.387}
SPL {X  -159.990, Y  +515.568, Z    +0.000, E1  +338.084, E3 -476964.484}
ENDSPLINE

SPLINE
SPL {X  -159.990, Y  +518.374, Z    +0.000, E1  +341.240, E3 -476977.072}
ENDSPLINE

SPLINE
SPL {X  -159.990, Y  +513.606, Z    +0.000, E1  +339.879, E3 -476992.983}
SPL {X  -159.990, Y  +508.660, Z    +0.000, E1  +338.515, E3 -477008.412}
SPL {X  -159.990, Y  +505.237, Z    +0.000, E1  +337.606, E3 -477018.669}
SPL {X  -159.990, Y  +501.963, Z    +0.000, E1  +336.712, E3 -477027.773}
SPL {X  -159.990, Y  +498.406, Z    +0.000, E1  +335.789, E3 -477037.524}
SPL {X  -159.990, Y  +494.693, Z    +0.000, E1  +334.929, E3 -477047.992}
SPL {X  -159.990, Y  +491.649, Z    +0.000, E1  +334.596, E3 -477059.194}
SPL {X  -159.990, Y  +488.807, Z    +0.000, E1  +334.603, E3 -477071.918}
SPL {X  -159.990, Y  +486.070, Z    +0.000, E1  +334.601, E3 -477084.149}
SPL {X  -159.990, Y  +483.747, Z    +0.000, E1  +334.616, E3 -477094.562}
SPL {X  -159.990, Y  +481.980, Z    +0.000, E1  +334.616, E3 -477102.460}
SPL {X  -159.990, Y  +479.252, Z    +0.000, E1  +334.588, E3 -477114.602}
SPL {X  -159.990, Y  +475.940, Z    +0.000, E1  +334.597, E3 -477129.422}
SPL {X  -159.990, Y  +473.026, Z    +0.000, E1  +334.601, E3 -477142.452}
SPL {X  -159.990, Y  +470.047, Z    +0.000, E1  +334.598, E3 -477155.770}
SPL {X  -159.990, Y  +466.213, Z    +0.000, E1  +334.567, E3 -477172.850}
SPL {X  -159.990, Y  +462.520, Z    +0.000, E1  +334.600, E3 -477189.418}
SPL {X  -159.990, Y  +460.081, Z    +0.000, E1  +334.610, E3 -477200.320}
SPL {X  -159.990, Y  +457.497, Z    +0.000, E1  +334.597, E3 -477211.844}
SPL {X  -159.990, Y  +455.126, Z    +0.000, E1  +334.611, E3 -477222.453}
SPL {X  -159.990, Y  +452.123, Z    +0.000, E1  +334.574, E3 -477235.810}
SPL {X  -159.990, Y  +448.503, Z    +0.000, E1  +334.590, E3 -477252.012}
SPL {X  -159.990, Y  +445.882, Z    +0.000, E1  +334.615, E3 -477263.814}
SPL {X  -159.990, Y  +443.345, Z    +0.000, E1  +334.610, E3 -477275.196}
SPL {X  -159.990, Y  +441.077, Z    +0.000, E1  +334.631, E3 -477285.395}
SPL {X  -159.990, Y  +438.608, Z    +0.000, E1  +334.608, E3 -477296.392}
SPL {X  -159.990, Y  +434.852, Z    +0.000, E1  +334.585, E3 -477313.146}
SPL {X  -159.990, Y  +430.645, Z    +0.000, E1  +334.586, E3 -477331.965}
SPL {X  -159.990, Y  +426.865, Z    +0.000, E1  +334.602, E3 -477348.895}
SPL {X  -159.990, Y  +424.251, Z    +0.000, E1  +334.625, E3 -477360.632}
SPL {X  -159.990, Y  +421.010, Z    +0.000, E1  +334.582, E3 -477375.047}
SPL {X  -159.990, Y  +417.103, Z    +0.000, E1  +334.600, E3 -477392.551}
SPL {X  -159.990, Y  +413.684, Z    +0.000, E1  +334.603, E3 -477407.850}
SPL {X  -159.990, Y  +410.645, Z    +0.000, E1  +334.615, E3 -477421.462}
SPL {X  -159.990, Y  +407.450, Z    +0.000, E1  +334.599, E3 -477435.710}
SPL {X  -159.990, Y  +403.513, Z    +0.000, E1  +334.580, E3 -477453.264}
SPL {X  -159.990, Y  +400.403, Z    +0.000, E1  +334.620, E3 -477467.246}
SPL {X  -159.990, Y  +397.743, Z    +0.000, E1  +334.600, E3 -477479.115}
SPL {X  -159.990, Y  +394.848, Z    +0.000, E1  +334.621, E3 -477492.117}
SPL {X  -159.990, Y  +392.473, Z    +0.000, E1  +334.623, E3 -477502.743}
SPL {X  -159.990, Y  +390.187, Z    +0.000, E1  +334.622, E3 -477513.001}
SPL {X  -159.990, Y  +387.503, Z    +0.000, E1  +334.622, E3 -477524.996}
SPL {X  -159.990, Y  +384.711, Z    +0.000, E1  +334.612, E3 -477537.440}
SPL {X  -159.988, Y  +381.794, Z    +0.000, E1  +334.611, E3 -477550.475}
SPL {X  -159.958, Y  +379.279, Z    +0.000, E1  +334.625, E3 -477561.765}
SPL {X  -159.894, Y  +376.959, Z    +0.000, E1  +334.630, E3 -477572.209}
SPL {X  -159.765, Y  +374.027, Z    +0.000, E1  +334.633, E3 -477585.425}
SPL {X  -159.607, Y  +371.442, Z    +0.000, E1  +334.673, E3 -477597.200}
SPL {X  -159.379, Y  +368.534, Z    +0.000, E1  +334.684, E3 -477610.387}
SPL {X  -159.113, Y  +365.767, Z    +0.000, E1  +334.734, E3 -477623.027}
SPL {X  -158.798, Y  +363.007, Z    +0.000, E1  +334.761, E3 -477635.667}
SPL {X  -158.453, Y  +360.380, Z    +0.000, E1  +334.828, E3 -477647.812}
SPL {X  -158.127, Y  +358.155, Z    +0.000, E1  +334.874, E3 -477658.143}
SPL {X  -158.095, Y  +357.947, Z    +0.000, E1  +338.259, E3 -477689.715}
ENDSPLINE

SPLINE
SPL {X  -158.454, Y  +360.384, Z    +0.000, E1  +340.634, E3 -477701.866}
SPL {X  -159.737, Y  +373.507, Z    +0.000, E1  +349.689, E3 -477723.901}
SPL {X  -159.990, Y  +382.574, Z    +0.000, E1  +355.537, E3 -477730.589}
SPL {X  -159.990, Y  +387.496, Z    +0.000, E1  +358.996, E3 -477733.334}
SPL {X  -159.990, Y  +395.121, Z    +0.000, E1  +364.514, E3 -477737.646}
SPL {X  -159.990, Y  +407.941, Z    +0.000, E1  +374.126, E3 -477749.721}
SPL {X  -159.990, Y  +418.671, Z    +0.000, E1  +379.855, E3 -477769.137}
SPL {X  -159.990, Y  +428.534, Z    +0.000, E1  +383.299, E3 -477792.657}
SPL {X  -159.990, Y  +431.017, Z    +0.000, E1  +383.339, E3 -477804.783}
SPL {X  -159.990, Y  +434.188, Z    +0.000, E1  +383.325, E3 -477820.407}
SPL {X  -159.990, Y  +437.007, Z    +0.000, E1  +383.323, E3 -477834.298}
SPL {X  -159.990, Y  +439.778, Z    +0.000, E1  +383.323, E3 -477847.931}
SPL {X  -159.990, Y  +442.945, Z    +0.000, E1  +383.339, E3 -477863.494}
SPL {X  -159.990, Y  +446.037, Z    +0.000, E1  +383.324, E3 -477878.745}
SPL {X  -159.990, Y  +448.341, Z    +0.000, E1  +383.317, E3 -477890.062}
SPL {X  -159.990, Y  +450.345, Z    +0.000, E1  +383.316, E3 -477899.940}
SPL {X  -159.990, Y  +452.828, Z    +0.000, E1  +383.330, E3 -477912.140}
SPL {X  -159.990, Y  +456.338, Z    +0.000, E1  +383.359, E3 -477929.332}
SPL {X  -159.990, Y  +459.480, Z    +0.000, E1  +383.323, E3 -477944.873}
SPL {X  -159.990, Y  +461.803, Z    +0.000, E1  +383.322, E3 -477956.308}
SPL {X  -159.990, Y  +464.971, Z    +0.000, E1  +383.357, E3 -477971.814}
SPL {X  -159.990, Y  +467.934, Z    +0.000, E1  +383.321, E3 -477986.472}
SPL {X  -159.990, Y  +469.939, Z    +0.000, E1  +383.319, E3 -477996.333}
SPL {X  -159.990, Y  +472.144, Z    +0.000, E1  +383.327, E3 -478007.184}
SPL {X  -159.990, Y  +474.152, Z    +0.000, E1  +383.309, E3 -478017.136}
SPL {X  -159.990, Y  +476.560, Z    +0.000, E1  +383.332, E3 -478028.944}
SPL {X  -159.990, Y  +478.770, Z    +0.000, E1  +383.306, E3 -478039.869}
SPL {X  -159.990, Y  +480.905, Z    +0.000, E1  +383.327, E3 -478050.337}
SPL {X  -159.990, Y  +484.251, Z    +0.000, E1  +383.352, E3 -478066.753}
SPL {X  -159.990, Y  +488.031, Z    +0.000, E1  +383.345, E3 -478085.386}
SPL {X  -159.990, Y  +491.121, Z    +0.000, E1  +383.323, E3 -478100.631}
SPL {X  -159.990, Y  +493.610, Z    +0.000, E1  +383.323, E3 -478112.884}
SPL {X  -159.990, Y  +496.863, Z    +0.000, E1  +383.350, E3 -478128.844}
SPL {X  -159.990, Y  +499.995, Z    +0.000, E1  +383.324, E3 -478144.306}
SPL {X  -159.990, Y  +502.341, Z    +0.000, E1  +383.320, E3 -478155.865}
SPL {X  -159.990, Y  +505.377, Z    +0.000, E1  +383.346, E3 -478170.755}
SPL {X  -159.990, Y  +508.697, Z    +0.000, E1  +383.335, E3 -478187.115}
SPL {X  -159.990, Y  +511.771, Z    +0.000, E1  +383.331, E3 -478202.262}
SPL {X  -159.990, Y  +514.016, Z    +0.000, E1  +383.308, E3 -478213.366}
SPL {X  -159.990, Y  +516.195, Z    +0.000, E1  +383.325, E3 -478224.053}
SPL {X  -159.990, Y  +518.925, Z    +0.000, E1  +383.333, E3 -478237.417}
SPL {X  -159.990, Y  +521.408, Z    +0.000, E1  +383.329, E3 -478249.626}
SPL {X  -159.990, Y  +523.942, Z    +0.000, E1  +383.333, E3 -478262.119}
SPL {X  -159.990, Y  +526.221, Z    +0.000, E1  +383.314, E3 -478273.395}
SPL {X  -159.990, Y  +527.834, Z    +0.000, E1  +383.311, E3 -478281.345}
SPL {X  -159.990, Y  +529.993, Z    +0.000, E1  +383.329, E3 -478291.920}
SPL {X  -159.990, Y  +532.441, Z    +0.000, E1  +383.322, E3 -478303.971}
SPL {X  -159.990, Y  +534.618, Z    +0.000, E1  +383.322, E3 -478314.704}
SPL {X  -159.990, Y  +537.024, Z    +0.000, E1  +383.321, E3 -478326.567}
SPL {X  -159.990, Y  +539.129, Z    +0.000, E1  +383.310, E3 -478336.950}
SPL {X  -159.990, Y  +541.183, Z    +0.000, E1  +383.319, E3 -478347.046}
SPL {X  -159.990, Y  +543.647, Z    +0.000, E1  +383.325, E3 -478359.149}
SPL {X  -159.990, Y  +545.957, Z    +0.000, E1  +383.318, E3 -478370.529}
SPL {X  -159.990, Y  +548.912, Z    +0.000, E1  +383.354, E3 -478384.989}
SPL {X  -159.990, Y  +551.655, Z    +0.000, E1  +383.320, E3 -478398.564}
SPL {X  -159.990, Y  +553.711, Z    +0.000, E1  +383.317, E3 -478408.686}
SPL {X  -159.990, Y  +556.481, Z    +0.000, E1  +383.354, E3 -478422.247}
SPL {X  -159.990, Y  +559.475, Z    +0.000, E1  +383.321, E3 -478437.053}
SPL {X  -159.990, Y  +561.830, Z    +0.000, E1  +383.325, E3 -478448.637}
SPL {X  -159.990, Y  +564.273, Z    +0.000, E1  +383.325, E3 -478460.662}
SPL {X  -159.990, Y  +566.342, Z    +0.000, E1  +383.314, E3 -478470.866}
SPL {X  -159.990, Y  +568.184, Z    +0.000, E1  +383.317, E3 -478479.927}
SPL {X  -159.990, Y  +570.314, Z    +0.000, E1  +383.326, E3 -478490.390}
SPL {X  -159.990, Y  +573.444, Z    +0.000, E1  +383.356, E3 -478505.729}
SPL {X  -159.990, Y  +576.445, Z    +0.000, E1  +383.320, E3 -478520.577}
SPL {X  -159.990, Y  +578.932, Z    +0.000, E1  +383.330, E3 -478532.794}
SPL {X  -159.990, Y  +581.497, Z    +0.000, E1  +383.329, E3 -478545.379}
SPL {X  -159.990, Y  +583.973, Z    +0.000, E1  +383.332, E3 -478557.564}
SPL {X  -159.990, Y  +586.020, Z    +0.000, E1  +383.323, E3 -478567.648}
SPL {X  -159.990, Y  +587.711, Z    +0.000, E1  +383.318, E3 -478575.988}
SPL {X  -159.990, Y  +589.763, Z    +0.000, E1  +383.328, E3 -478586.064}
SPL {X  -159.990, Y  +591.698, Z    +0.000, E1  +383.324, E3 -478595.548}
SPL {X  -159.990, Y  +593.847, Z    +0.000, E1  +383.340, E3 -478606.079}
SPL {X  -159.990, Y  +597.018, Z    +0.000, E1  +383.367, E3 -478621.611}
SPL {X  -159.990, Y  +599.887, Z    +0.000, E1  +383.341, E3 -478635.715}
SPL {X  -159.990, Y  +601.949, Z    +0.000, E1  +383.344, E3 -478645.842}
SPL {X  -159.990, Y  +605.106, Z    +0.000, E1  +383.383, E3 -478661.288}
SPL {X  -159.990, Y  +608.111, Z    +0.000, E1  +383.342, E3 -478676.139}
SPL {X  -159.990, Y  +610.073, Z    +0.000, E1  +383.343, E3 -478685.797}
SPL {X  -159.990, Y  +612.330, Z    +0.000, E1  +383.340, E3 -478696.925}
SPL {X  -159.990, Y  +615.036, Z    +0.000, E1  +383.353, E3 -478710.212}
SPL {X  -159.990, Y  +618.481, Z    +0.000, E1  +383.366, E3 -478727.150}
SPL {X  -159.990, Y  +621.517, Z    +0.000, E1  +383.337, E3 -478742.133}
SPL {X  -159.990, Y  +623.764, Z    +0.000, E1  +383.335, E3 -478753.183}
SPL {X  -159.990, Y  +626.608, Z    +0.000, E1  +383.361, E3 -478767.108}
SPL {X  -159.990, Y  +630.271, Z    +0.000, E1  +383.375, E3 -478785.069}
SPL {X  -159.990, Y  +633.318, Z    +0.000, E1  +383.339, E3 -478800.147}
SPL {X  -159.990, Y  +635.650, Z    +0.000, E1  +383.339, E3 -478811.618}
SPL {X  -159.990, Y  +638.406, Z    +0.000, E1  +383.354, E3 -478825.184}
SPL {X  -159.990, Y  +641.831, Z    +0.000, E1  +383.342, E3 -478842.132}
SPL {X  -159.990, Y  +644.884, Z    +0.000, E1  +383.324, E3 -478857.219}
SPL {X  -159.990, Y  +647.550, Z    +0.000, E1  +383.318, E3 -478870.386}
SPL {X  -159.990, Y  +650.790, Z    +0.000, E1  +383.346, E3 -478886.252}
SPL {X  -159.990, Y  +654.543, Z    +0.000, E1  +383.348, E3 -478904.705}
SPL {X  -159.990, Y  +658.319, Z    +0.000, E1  +383.349, E3 -478923.295}
SPL {X  -159.990, Y  +661.392, Z    +0.000, E1  +383.318, E3 -478938.498}
SPL {X  -159.990, Y  +663.662, Z    +0.000, E1  +383.322, E3 -478949.622}
SPL {X  -159.990, Y  +665.964, Z    +0.000, E1  +383.328, E3 -478960.912}
SPL {X  -159.990, Y  +667.870, Z    +0.000, E1  +383.320, E3 -478970.319}
SPL {X  -159.990, Y  +669.861, Z    +0.000, E1  +383.321, E3 -478980.120}
SPL {X  -159.990, Y  +671.893, Z    +0.000, E1  +383.319, E3 -478990.128}
SPL {X  -159.974, Y  +673.789, Z    +0.000, E1  +383.323, E3 -478999.444}
SPL {X  -159.924, Y  +676.110, Z    +0.000, E1  +383.320, E3 -479010.929}
SPL {X  -159.801, Y  +679.265, Z    +0.000, E1  +383.327, E3 -479026.547}
SPL {X  -159.626, Y  +682.287, Z    +0.000, E1  +383.280, E3 -479041.646}
SPL {X  -159.462, Y  +684.486, Z    +0.000, E1  +383.258, E3 -479052.645}
SPL {X  -159.212, Y  +687.262, Z    +0.000, E1  +383.238, E3 -479066.549}
SPL {X  -158.971, Y  +689.529, Z    +0.000, E1  +383.181, E3 -479078.009}
SPL {X  -158.658, Y  +692.098, Z    +0.000, E1  +383.176, E3 -479090.915}
ENDSPLINE

SPLINE
SPL {X  -159.063, Y  +688.696, Z    +0.000, E1  +377.094, E3 -479133.134}
SPL {X  -159.987, Y  +672.488, Z    +0.000, E1  +365.638, E3 -479157.199}
SPL {X  -159.990, Y  +663.928, Z    +0.000, E1  +359.662, E3 -479162.994}
SPL {X  -159.990, Y  +658.009, Z    +0.000, E1  +355.226, E3 -479166.693}
SPL {X  -159.990, Y  +651.879, Z    +0.000, E1  +350.548, E3 -479171.756}
SPL {X  -159.990, Y  +639.151, Z    +0.000, E1  +342.343, E3 -479186.991}
SPL {X  -159.990, Y  +635.956, Z    +0.000, E1  +340.738, E3 -479192.676}
SPL {X  -159.990, Y  +626.634, Z    +0.000, E1  +337.968, E3 -479220.200}
SPL {X  -159.990, Y  +624.622, Z    +0.000, E1  +337.980, E3 -479230.784}
SPL {X  -159.990, Y  +622.489, Z    +0.000, E1  +337.969, E3 -479241.950}
SPL {X  -159.990, Y  +619.955, Z    +0.000, E1  +337.968, E3 -479255.240}
SPL {X  -159.990, Y  +617.386, Z    +0.000, E1  +337.968, E3 -479268.715}
SPL {X  -159.990, Y  +614.863, Z    +0.000, E1  +337.969, E3 -479281.947}
SPL {X  -159.990, Y  +612.600, Z    +0.000, E1  +337.975, E3 -479293.831}
SPL {X  -159.990, Y  +610.646, Z    +0.000, E1  +337.979, E3 -479304.089}
SPL {X  -159.990, Y  +608.810, Z    +0.000, E1  +337.977, E3 -479313.722}
SPL {X  -159.990, Y  +605.804, Z    +0.000, E1  +337.936, E3 -479329.367}
SPL {X  -159.990, Y  +602.819, Z    +0.000, E1  +337.963, E3 -479345.038}
SPL {X  -159.990, Y  +600.642, Z    +0.000, E1  +337.968, E3 -479356.466}
SPL {X  -159.990, Y  +598.568, Z    +0.000, E1  +337.954, E3 -479367.259}
SPL {X  -159.990, Y  +596.440, Z    +0.000, E1  +337.964, E3 -479378.440}
SPL {X  -159.990, Y  +593.768, Z    +0.000, E1  +337.929, E3 -479392.373}
SPL {X  -159.990, Y  +590.068, Z    +0.000, E1  +337.924, E3 -479411.742}
SPL {X  -159.990, Y  +586.620, Z    +0.000, E1  +337.935, E3 -479429.804}
SPL {X  -159.990, Y  +584.080, Z    +0.000, E1  +337.953, E3 -479443.131}
SPL {X  -159.990, Y  +581.924, Z    +0.000, E1  +337.949, E3 -479454.431}
SPL {X  -159.990, Y  +578.886, Z    +0.000, E1  +337.918, E3 -479470.285}
SPL {X  -159.990, Y  +576.252, Z    +0.000, E1  +337.962, E3 -479484.183}
SPL {X  -159.990, Y  +574.188, Z    +0.000, E1  +337.947, E3 -479494.956}
SPL {X  -159.990, Y  +571.954, Z    +0.000, E1  +337.959, E3 -479506.713}
SPL {X  -159.990, Y  +570.110, Z    +0.000, E1  +337.958, E3 -479516.364}
SPL {X  -159.990, Y  +568.165, Z    +0.000, E1  +337.957, E3 -479526.544}
SPL {X  -159.990, Y  +566.106, Z    +0.000, E1  +337.954, E3 -479537.327}
SPL {X  -159.990, Y  +563.259, Z    +0.000, E1  +337.929, E3 -479552.209}
SPL {X  -159.990, Y  +559.661, Z    +0.000, E1  +337.922, E3 -479571.031}
SPL {X  -159.990, Y  +555.965, Z    +0.000, E1  +337.915, E3 -479590.340}
SPL {X  -159.990, Y  +553.115, Z    +0.000, E1  +337.946, E3 -479605.326}
SPL {X  -159.990, Y  +550.886, Z    +0.000, E1  +337.944, E3 -479617.007}
SPL {X  -159.990, Y  +548.568, Z    +0.000, E1  +337.944, E3 -479629.129}
SPL {X  -159.990, Y  +545.859, Z    +0.000, E1  +337.926, E3 -479643.278}
SPL {X  -159.990, Y  +542.390, Z    +0.000, E1  +337.914, E3 -479661.449}
SPL {X  -159.990, Y  +539.341, Z    +0.000, E1  +337.944, E3 -479677.470}
SPL {X  -159.990, Y  +536.935, Z    +0.000, E1  +337.942, E3 -479690.060}
SPL {X  -159.990, Y  +534.656, Z    +0.000, E1  +337.946, E3 -479702.003}
SPL {X  -159.990, Y  +531.679, Z    +0.000, E1  +337.913, E3 -479717.517}
SPL {X  -159.990, Y  +527.941, Z    +0.000, E1  +337.907, E3 -479737.060}
SPL {X  -159.990, Y  +525.053, Z    +0.000, E1  +337.942, E3 -479752.250}
SPL {X  -159.990, Y  +522.838, Z    +0.000, E1  +337.933, E3 -479763.854}
SPL {X  -159.990, Y  +519.698, Z    +0.000, E1  +337.916, E3 -479780.237}
SPL {X  -159.990, Y  +517.251, Z    +0.000, E1  +337.946, E3 -479793.097}
SPL {X  -159.990, Y  +515.568, Z    +0.000, E1  +338.084, E3 -479803.194}
ENDSPLINE

SPLINE
SPL {X  -159.990, Y  +517.293, Z    +0.000, E1  +340.923, E3 -479819.492}
ENDSPLINE

SPLINE
SPL {X  -159.990, Y  +512.548, Z    +0.000, E1  +339.587, E3 -479835.067}
SPL {X  -159.990, Y  +508.660, Z    +0.000, E1  +338.515, E3 -479847.122}
SPL {X  -159.990, Y  +503.499, Z    +0.000, E1  +337.116, E3 -479862.201}
SPL {X  -159.990, Y  +498.406, Z    +0.000, E1  +335.789, E3 -479876.234}
SPL {X  -159.990, Y  +494.693, Z    +0.000, E1  +334.929, E3 -479886.701}
SPL {X  -159.990, Y  +491.649, Z    +0.000, E1  +334.596, E3 -479897.904}
SPL {X  -159.990, Y  +488.807, Z    +0.000, E1  +334.603, E3 -479910.628}
SPL {X  -159.990, Y  +486.070, Z    +0.000, E1  +334.601, E3 -479922.859}
SPL {X  -159.990, Y  +483.747, Z    +0.000, E1  +334.616, E3 -479933.272}
SPL {X  -159.990, Y  +481.038, Z    +0.000, E1  +334.588, E3 -479945.327}
SPL {X  -159.990, Y  +477.508, Z    +0.000, E1  +334.590, E3 -479961.110}
SPL {X  -159.990, Y  +473.634, Z    +0.000, E1  +334.574, E3 -479978.399}
SPL {X  -159.990, Y  +470.047, Z    +0.000, E1  +334.598, E3 -479994.480}
SPL {X  -159.990, Y  +467.082, Z    +0.000, E1  +334.601, E3 -480007.727}
SPL {X  -159.990, Y  +464.919, Z    +0.000, E1  +334.619, E3 -480017.454}
SPL {X  -159.990, Y  +462.520, Z    +0.000, E1  +334.600, E3 -480028.128}
SPL {X  -159.990, Y  +460.081, Z    +0.000, E1  +334.610, E3 -480039.029}
SPL {X  -159.990, Y  +457.497, Z    +0.000, E1  +334.597, E3 -480050.554}
SPL {X  -159.990, Y  +454.323, Z    +0.000, E1  +334.588, E3 -480064.713}
SPL {X  -159.990, Y  +450.823, Z    +0.000, E1  +334.583, E3 -480080.342}
SPL {X  -159.990, Y  +447.982, Z    +0.000, E1  +334.607, E3 -480093.082}
SPL {X  -159.990, Y  +445.108, Z    +0.000, E1  +334.593, E3 -480105.959}
SPL {X  -159.990, Y  +441.797, Z    +0.000, E1  +334.610, E3 -480120.838}
SPL {X  -159.990, Y  +439.442, Z    +0.000, E1  +334.631, E3 -480131.416}
SPL {X  -159.990, Y  +436.316, Z    +0.000, E1  +334.580, E3 -480145.298}
SPL {X  -159.990, Y  +432.613, Z    +0.000, E1  +334.610, E3 -480161.923}
SPL {X  -159.990, Y  +429.827, Z    +0.000, E1  +334.620, E3 -480174.400}
SPL {X  -159.990, Y  +426.865, Z    +0.000, E1  +334.602, E3 -480187.605}
SPL {X  -159.990, Y  +423.417, Z    +0.000, E1  +334.600, E3 -480203.021}
SPL {X  -159.990, Y  +420.283, Z    +0.000, E1  +334.614, E3 -480217.065}
SPL {X  -159.990, Y  +417.103, Z    +0.000, E1  +334.600, E3 -480231.260}
SPL {X  -159.990, Y  +413.684, Z    +0.000, E1  +334.603, E3 -480246.559}
SPL {X  -159.990, Y  +410.645, Z    +0.000, E1  +334.615, E3 -480260.171}
SPL {X  -159.990, Y  +408.351, Z    +0.000, E1  +334.628, E3 -480270.457}
SPL {X  -159.990, Y  +406.574, Z    +0.000, E1  +334.625, E3 -480278.374}
SPL {X  -159.990, Y  +404.255, Z    +0.000, E1  +334.609, E3 -480288.711}
SPL {X  -159.990, Y  +401.103, Z    +0.000, E1  +334.596, E3 -480302.775}
SPL {X  -159.990, Y  +398.389, Z    +0.000, E1  +334.619, E3 -480314.971}
SPL {X  -159.990, Y  +395.411, Z    +0.000, E1  +334.600, E3 -480328.268}
SPL {X  -159.990, Y  +392.473, Z    +0.000, E1  +334.623, E3 -480341.453}
SPL {X  -159.990, Y  +390.187, Z    +0.000, E1  +334.622, E3 -480351.711}
SPL {X  -159.990, Y  +387.503, Z    +0.000, E1  +334.622, E3 -480363.706}
SPL {X  -159.990, Y  +384.711, Z    +0.000, E1  +334.612, E3 -480376.150}
SPL {X  -159.988, Y  +381.794, Z    +0.000, E1  +334.611, E3 -480389.184}
SPL {X  -159.958, Y  +379.279, Z    +0.000, E1  +334.625, E3 -480400.475}
SPL {X  -159.894, Y  +376.959, Z    +0.000, E1  +334.630, E3 -480410.919}
SPL {X  -159.765, Y  +374.027, Z    +0.000, E1  +334.633, E3 -480424.135}
SPL {X  -159.607, Y  +371.442, Z    +0.000, E1  +334.673, E3 -480435.910}
SPL {X  -159.379, Y  +368.534, Z    +0.000, E1  +334.684, E3 -480449.097}
SPL {X  -159.113, Y  +365.767, Z    +0.000, E1  +334.734, E3 -480461.737}
SPL {X  -158.798, Y  +363.007, Z    +0.000, E1  +334.761, E3 -480474.377}
SPL {X  -158.453, Y  +360.380, Z    +0.000, E1  +334.828, E3 -480486.521}
SPL {X  -158.127, Y  +358.155, Z    +0.000, E1  +334.874, E3 -480496.852}
SPL {X  -158.095, Y  +357.947, Z    +0.000, E1  +338.259, E3 -480528.425}
ENDSPLINE

